// TIA Portal project "ContainerProduction_V0.1.0" (V18)

(* hardware
DEVICE "S7-1500/ET200MP station_1"  S7-1500 station
   slot 0: "Rail_0"  Rack  6ES7 590-1***0-0AA0
   slot 1: "PLC_1"  CPU 1511C-1 PN  6ES7 511-1CK01-0AB0  V2.9
      slot 3: "CPU display_1"  6ES7591-1AA00-0AA0
      slot 32768: "PROFINET interface_1"  X1
         slot 32769: "Port_1"  X1 P1
         slot 32770: "Port_2"  X1 P2
      slot 34817: "Virtual CP interface port_1"  Virtual CP interface port  Virtual CP interface port
*)

// ===== PLC "PLC_1"  CPU 1511C-1 PN =====

VAR_GLOBAL   // PLC tag table "Default tag table"
   "start_btn_sim" AT %M501.0 : Bool;
   "stp_btn_sim" AT %M501.1 : Bool;
   "monitor1 state value" AT %MW2 : UInt;
   "Spare_memory2" AT %M500.2 : Bool;
   "Spare_memory1" AT %M500.3 : Bool;
   "Spare_memory3" AT %M500.4 : Bool;
   "Spare_memory5" AT %M500.5 : Bool;
   "Tag_3" AT %M500.6 : Bool;
   "Tag_4" AT %M500.7 : Bool;
   "Tag_5" AT %M500.1 : Bool;
   "Tag_6" AT %M501.2 : Bool;
   "Tag_7" AT %M111.7 : Bool;
   "Tag_8" AT %M856.7 : Bool;
   "Tag_9" AT %M358.7 : Bool;
   "Tag_10" AT %M123.4 : Bool;
   "Clock_Byte" AT %MB0 : Byte;
   "Clock_10Hz" AT %M0.0 : Bool;
   "Clock_5Hz" AT %M0.1 : Bool;
   "Clock_2.5Hz" AT %M0.2 : Bool;
   "Clock_2Hz" AT %M0.3 : Bool;
   "Clock_1.25Hz" AT %M0.4 : Bool;
   "Clock_1Hz" AT %M0.5 : Bool;
   "Clock_0.625Hz" AT %M0.6 : Bool;
   "Clock_0.5Hz" AT %M0.7 : Bool;
   "Tag_1" AT %M525.5 : Bool;
   "index" AT %MW4 : UInt;   // actual array index value
   "Tag_2" AT %M503.7 : Bool;
   "Tag_11" AT %M853.7 : Bool;
   "Tag_12" AT %M853.0 : Bool;
   "Tag_13" AT %M444.0 : Bool;
END_VAR

VAR_GLOBAL   // PLC tag table "IO_List"
   "Start_Button" AT %I10.0 : Bool;
   "Stop_Button" AT %I10.1 : Bool;
   "Emergency_Stop" AT %I10.2 : Bool;
   "Mold_isClosed" AT %I10.3 : Bool;
   "Mold_isOpen" AT %I10.4 : Bool;
   "Product_Ejected" AT %I10.7 : Bool;
   "NextStation_Buffer_Full" AT %I11.0 : Bool;
   "DI_unused1" AT %I11.1 : Bool;
   "Feeder_Start" AT %Q4.0 : Bool;
   "Injection_Start" AT %Q4.1 : Bool;
   "Mold_Close" AT %Q4.2 : Bool;
   "Mold_Open" AT %Q4.3 : Bool;
   "Ejector_Forward" AT %Q4.4 : Bool;
   "Ejector_Backward" AT %Q4.5 : Bool;
   "Heater_Enable" AT %Q4.6 : Bool;
   "Cooling_Enable" AT %Q4.7 : Bool;
   "Alarm_Buzzer" AT %Q5.0 : Bool;
   "Tower_Light_Red" AT %Q5.1 : Bool;
   "Material_ActLevel" AT %IW0 : Word;
   "Temperature_ActLevel" AT %IW2 : Word;
   "Air_Pressure_ActLevel" AT %IW4 : Word;
   "AQ_unused1" AT %QW0 : Word;
   "Ejector_is_atHome" AT %I10.5 : Bool;
   "Ejector_isExtended" AT %I10.6 : Bool;
   "DI_unused2" AT %I11.2 : Bool;
   "DI_unused3" AT %I11.3 : Bool;
   "DI_unused4" AT %I11.4 : Bool;
   "DI_unused5" AT %I11.5 : Bool;
   "DI_unused6" AT %I11.6 : Bool;
   "DI_unused7" AT %I11.7 : Bool;
   "Tower_Light_Yellow" AT %Q5.2 : Bool;
   "Tower_Light_Green" AT %Q5.3 : Bool;
   "Goto_NextStationBuffer" AT %Q5.4 : Bool;
   "DQ_unused1" AT %Q5.5 : Bool;
   "DQ_unused2" AT %Q5.6 : Bool;
   "DQ_unused3" AT %Q5.7 : Bool;
   "AI_unused1" AT %IW6 : Word;
   "AI_unused2" AT %IW8 : Word;
   "AQ_unused2" AT %QW2 : Word;
END_VAR

// folder: Config

DATA_BLOCK "config_parameters"   // DB2
{ S7_Optimized_Access := 'TRUE' }
VERSION : 0.1
   VAR
      Receipe_Parameters : Array[0..100] of Struct
         Heating_Time : Time;
         Cooling_Time : Time;
         Material_Consumption : Real;
         Temperature_SetVal : Real;
         Pressure_SetVal : Real;
      END_STRUCT;
      Station_Parameters : Struct
         Hopper : Struct
            ErrorLimit : Real := 1250.0;
            HighLimit : Real := 1000.0;
            LowLimit : Real := 350.0;
            EmptyLimit : Real := 50.0;
         END_STRUCT;
         Temperature : Struct
            ErrorLimit : Real := 600.0;
            HighLimit : Real := 550.0;
            LowLimit : Real := 400.0;
         END_STRUCT;
         Pressure : Struct
            ErrorLimit : Real := 15.0;
            HighLimit : Real := 13.0;
            LowLimit : Real := 10.0;
         END_STRUCT;
         Timeout : Struct
            Mold : Struct
               Open : Time;
               Close : Time;
            END_STRUCT;
            Ejector : Struct
               Open : Time;
               Close : Time;
            END_STRUCT;
            ProductDetect : Time;
            Transfer : Time;
         END_STRUCT;
      END_STRUCT;
   END_VAR
BEGIN
   Receipe_Parameters[2].Pressure_SetVal := 12.0;
   Receipe_Parameters[2].Temperature_SetVal := 525.0;
   Receipe_Parameters[2].Material_Consumption := 2000.0;
   Receipe_Parameters[1].Pressure_SetVal := 11.5;   // Pressure_SetVal
   Receipe_Parameters[1].Temperature_SetVal := 500.0;   // Temperature_SetVal
   Receipe_Parameters[1].Material_Consumption := 1000.0;   // Material_Consumption
   Receipe_Parameters[1].Cooling_Time := T#7S;   // Cooling_Time
   Receipe_Parameters[2].Cooling_Time := T#13S;
   Receipe_Parameters[1].Heating_Time := T#5S;   // Heating_Time
   Receipe_Parameters[2].Heating_Time := T#10S;
   Receipe_Parameters[0].Heating_Time := T#3S;
   Receipe_Parameters[0].Cooling_Time := T#3S;
   Receipe_Parameters[0].Material_Consumption := 500.0;
   Receipe_Parameters[0].Temperature_SetVal := 450.0;
   Receipe_Parameters[0].Pressure_SetVal := 11.0;
END_DATA_BLOCK

// folder: Flow-1_Checking_Order_Data

DATA_BLOCK "FB_create_serialNo_DB"   // DB8
{ S7_Optimized_Access := 'TRUE' }
VERSION : 0.1
// stored: InstanceOfName FB_create_serialNo
"FB_create_serialNo"
BEGIN
END_DATA_BLOCK

DATA_BLOCK "FB_CheckOrderData_DB"   // DB23
{ S7_Optimized_Access := 'TRUE' }
VERSION : 0.1
// stored: InstanceOfName FB_CheckOrderData
"FB_CheckOrderData"
BEGIN
END_DATA_BLOCK

// folder: Flow-1_Checking_Order_Data/Checking_MES_data

DATA_BLOCK "FB_checking_orderID_DB_1"   // DB12
{ S7_Optimized_Access := 'TRUE' }
VERSION : 0.1
// stored: InstanceOfName FB_checking_orderID
"FB_checking_orderID"
BEGIN
END_DATA_BLOCK

DATA_BLOCK "FB_checking_productID_DB_1"   // DB13
{ S7_Optimized_Access := 'TRUE' }
VERSION : 0.1
// stored: InstanceOfName FB_checking_productID
"FB_checking_productID"
BEGIN
END_DATA_BLOCK

DATA_BLOCK "FB_checking_receipeID_DB_1"   // DB14
{ S7_Optimized_Access := 'TRUE' }
VERSION : 0.1
// stored: InstanceOfName FB_checking_receipeID
"FB_checking_receipeID"
BEGIN
END_DATA_BLOCK

// folder: Flow-2_Checking_Initial_Conditions

DATA_BLOCK "FB_Control_Initial_Conditions_DB"   // DB25
{ S7_Optimized_Access := 'TRUE' }
VERSION : 0.1
// stored: InstanceOfName FB_Control_Initial_Conditions
"FB_Control_Initial_Conditions"
BEGIN
END_DATA_BLOCK

// folder: Flow3_Run_Molding_State

DATA_BLOCK "FB_Start_Molding_State_DB"   // DB11
{ S7_Optimized_Access := 'TRUE' }
VERSION : 0.1
// stored: InstanceOfName FB_Start_Molding_State
"FB_Start_Molding_State"
BEGIN
END_DATA_BLOCK

// folder: Flow4_Finishing_Molding_State

DATA_BLOCK "FB_Finishing_Molding_DB"   // DB15
{ S7_Optimized_Access := 'TRUE' }
VERSION : 0.1
// stored: InstanceOfName FB_Finishing_Molding
"FB_Finishing_Molding"
BEGIN
END_DATA_BLOCK

// folder: Flow5_Checking_Target_Production

DATA_BLOCK "FB_Checking_Target_Production_DB"   // DB16
{ S7_Optimized_Access := 'TRUE' }
VERSION : 0.1
// stored: InstanceOfName FB_Checking_Target_Production
"FB_Checking_Target_Production"
BEGIN
END_DATA_BLOCK

// folder: Machine_transition

DATA_BLOCK "FB_SubTransition_DB"   // DB9
{ S7_Optimized_Access := 'TRUE' }
VERSION : 0.1
// stored: InstanceOfName FB_SubTransition
"FB_SubTransition"
BEGIN
END_DATA_BLOCK

DATA_BLOCK "FB_control_state_transition_DB"   // DB10
{ S7_Optimized_Access := 'TRUE' }
VERSION : 0.1
// stored: InstanceOfName FB_control_state_transition
"FB_control_state_transition"
BEGIN
END_DATA_BLOCK

// folder: Simulation_data

DATA_BLOCK "FB_simulate_digital_input_DB"   // DB7
{ S7_Optimized_Access := 'TRUE' }
VERSION : 0.1
// stored: InstanceOfName FB_simulate_digital_input
"FB_simulate_digital_input"
BEGIN
END_DATA_BLOCK

DATA_BLOCK "Material_ActLevel_Simulation"   // DB18
{ S7_Optimized_Access := 'TRUE' }
VERSION : 0.1
// stored: InstanceOfName FB_simulate_analog_data
"FB_simulate_analog_data"
BEGIN
END_DATA_BLOCK

DATA_BLOCK "Temperature_Act_Level_Simulation"   // DB19
{ S7_Optimized_Access := 'TRUE' }
VERSION : 0.1
// stored: InstanceOfName FB_simulate_analog_data
"FB_simulate_analog_data"
BEGIN
END_DATA_BLOCK

DATA_BLOCK "Pressure_Act_Level_Simulation"   // DB20
{ S7_Optimized_Access := 'TRUE' }
VERSION : 0.1
// stored: InstanceOfName FB_simulate_analog_data
"FB_simulate_analog_data"
BEGIN
END_DATA_BLOCK

DATA_BLOCK "FB_simulate_digital_input_DB_1"   // DB24
{ S7_Optimized_Access := 'TRUE' }
VERSION : 0.1
// stored: InstanceOfName FB_simulate_digital_input
"FB_simulate_digital_input"
BEGIN
END_DATA_BLOCK

// folder: System blocks/Program resources

DATA_BLOCK "IEC_Counter_0_DB"   // DB17
{ S7_Optimized_Access := 'TRUE' }
AUTHOR : Simatic
FAMILY : IEC
NAME : CNTR
VERSION : 1.0
// stored: InstanceOfName IEC_COUNTER
"IEC_COUNTER"
BEGIN
END_DATA_BLOCK

DATA_BLOCK "IEC_Counter_0_DB_1"   // DB21
{ S7_Optimized_Access := 'TRUE' }
AUTHOR : Simatic
FAMILY : IEC
NAME : UCNTR
VERSION : 1.2
// stored: InstanceOfName IEC_UCOUNTER
"IEC_UCOUNTER"
BEGIN
END_DATA_BLOCK

DATA_BLOCK "IEC_Counter_0_DB_2"   // DB22
{ S7_Optimized_Access := 'TRUE' }
AUTHOR : Simatic
FAMILY : IEC
NAME : CNTR
VERSION : 1.0
// stored: InstanceOfName IEC_COUNTER
"IEC_COUNTER"
BEGIN
END_DATA_BLOCK

// folder: Variable

DATA_BLOCK "VAR_input_simulation"   // DB1
{ S7_Optimized_Access := 'TRUE' }
VERSION : 0.1
   VAR
      DI : Struct
         Start_Button : Bool;
         Stop_Button : Bool;
         Emergency_Stop : Bool;
         Mold_isClosed : Bool;
         Mold_isOpen : Bool := true;
         Ejector_is_atHome : Bool := true;
         Ejector_isExtended : Bool;
         Product_Ejected : Bool;
         NextStation_Buffer_Full : Bool;
         DI_unused1 : Bool := true;
         DI_unused2 : Bool := true;
         DI_unused3 : Bool := true;
         DI_unused4 : Bool := true;
         DI_unused5 : Bool := true;
         DI_unused6 : Bool := true;
         DI_unused7 : Bool := true;
      END_STRUCT;
      AI : Struct
         Material_ActLevel : Real;
         Temperature_ActLevel : Real;
         Air_Pressure_ActLevel : Real;
         AI_unused1 : Real;
         AI_unused2 : Real;
      END_STRUCT;
      Man_material_filling : Bool;
   END_VAR
BEGIN
END_DATA_BLOCK

DATA_BLOCK "VAR_Mes_to_ProductionLine"   // DB3
{ S7_Optimized_Access := 'TRUE' }
VERSION : 0.1
   VAR
      is_Order_Valid : Bool;
      Start_Order : Bool;
      received_MES_data : Struct
         OrderID : String := 'ORD-2026-4321';
         ProductID : String := 'CAP-05L';
         ReciepeID : String := 'RCP-001';
         TargetQuantity : UInt := 500;
      END_STRUCT;
      transmit_MES_data : Struct
         ProductInfo : Struct
            OrderID : String;
            ProductID : UInt;
            ReciepeID : UInt;
            TargetQuantity : UInt;
            ProductSerialNo : String;
         END_STRUCT;
         StationInfo : Struct
            StateNo : UInt;
            StateDescription : String;
            ErrorCode : UInt;
            ErrorDescription : String;
            WarningCode : UInt;
            WarninDescription : String;
            TotalProductionTime : Time;
            ProducedCount : UInt;
            OrderCompleted : Bool;
         END_STRUCT;
         ActualMeasurements : Struct
            ActualTemperature : Real;
            ActualPressure : Real;
            ActualHopperWeight : Real;
         END_STRUCT;
      END_STRUCT;
   END_VAR
BEGIN
END_DATA_BLOCK

DATA_BLOCK "VAR_state_machine"   // DB4
{ S7_Optimized_Access := 'TRUE' }
VERSION : 0.1
   VAR
      start_request : Bool;
      stop_request : Bool;
      st_idle : UInt := 0;
      st_checking_order : UInt := 100;
      st_checking_initial_safety : UInt := 200;
      st_running_molding : UInt := 300;
      st_finishing_molding : UInt := 400;
      st_cycle_completed : UInt := 500;
      st_checking_order_target : UInt := 600;
      st_order_finishing : UInt := 700;
      st_fault : UInt := 9999;
      st_machine_state : UInt := 0;
      previous_state_done : Bool;
      st_simulation_timers : Array[0..5] of IEC_TIMER;
   END_VAR
BEGIN
   st_simulation_timers[0].PT := T#2S_500MS;
   st_simulation_timers[1].PT := T#300MS;
   st_simulation_timers[2].PT := T#1s;
END_DATA_BLOCK

DATA_BLOCK "VAR_outputs"   // DB5
{ S7_Optimized_Access := 'TRUE' }
VERSION : 0.1
   VAR
      Feeder_Start : Bool;
      Injection_Start : Bool;
      Mold_Close : Bool;
      Mold_Open : Bool;
      Ejector_Forward : Bool;
      Ejector_Backward : Bool;
      Heater_Enable : Bool;
      Cooling_Enable : Bool;
      Alarm_Buzzer : Bool;
      Tower_Light_Red : Bool;
      Tower_Light_Yellow : Bool;
      Tower_Light_Green : Bool;
      Goto_NextStationBuffer : Bool;
      DQ_unused1 : Bool;
      DQ_unused2 : Bool;
      DQ_unused3 : Bool;
      AQ_unused1 : Real;
      AQ_unused2 : Real;
   END_VAR
BEGIN
END_DATA_BLOCK

DATA_BLOCK "Err_Wrn_list"   // DB6
{ S7_Optimized_Access := 'TRUE' }
VERSION : 0.1
   VAR
      error_active : Bool;
      warning_active : Bool;
      error_value : UInt;
      warning_value : UInt;
      error_list : Array[0..99] of String;
      warning_list : Array[0..99] of String;
   END_VAR
BEGIN
   error_list[0] := 'No Error';   // Emergeny stop is activated
   error_list[1] := 'Stop request is received';   // Mold is open
   error_list[2] := 'Received OrderID is invalid.';   // Material tank is empty
   error_list[3] := 'Received ProductID is invalid.';   // Thermal value is out of range
   error_list[5] := 'Received target production quantity is invalid.';   // Safety gurad is open
   error_list[4] := 'Received ReceipeID is invalid.';   // Pressure value is out of range
   error_list[6] := 'Creating serialNo error';   // Invalid OrderID
   warning_list[0] := 'No Warning';   // Stop request is received
   warning_list[1] := 'Raw material level is low. Feeding in progress.';   // Material level is low
   error_list[7] := 'Raw material level is too high.';   // Invalid ProductID
   error_list[8] := 'Actual Pressure value is low.';   // Invalid ReceipeID
   error_list[9] := 'Actual pressure level is too high.';   // Invalid Quantity
   error_list[10] := 'Mold closing error';
   error_list[11] := 'Ejector is not at home.';
   error_list[12] := 'Next station buffer is full';
   warning_list[2] := 'Raw material level is critic. Feeding in progress.';
   error_list[13] := 'Temperature is too high.';
   error_list[14] := 'Mold opening error';
END_DATA_BLOCK

// folder: (top level)

FUNCTION_BLOCK "backup"   // FB14, LAD
{ S7_Optimized_Access := 'TRUE' }
VERSION : 0.1
   VAR_TEMP
      Act_rcp_data : UInt;
   END_VAR
BEGIN

REGION Network 1 (SCL): Find out actual receipe parameters in config data
   IF "VAR_Mes_to_ProductionLine".transmit_MES_data.ProductInfo.ProductID <> 0 THEN
       IF "VAR_Mes_to_ProductionLine".transmit_MES_data.ProductInfo.ReciepeID <> 0 THEN
           "index" := "VAR_Mes_to_ProductionLine".transmit_MES_data.ProductInfo.ReciepeID - 1;
           //#Act_rcp_data := "config_parameters".Receipe_Parameters["index"];
       END_IF;
   END_IF;
END_REGION

REGION Network 2: Simulate Analog Inputs according to reciepe parameters
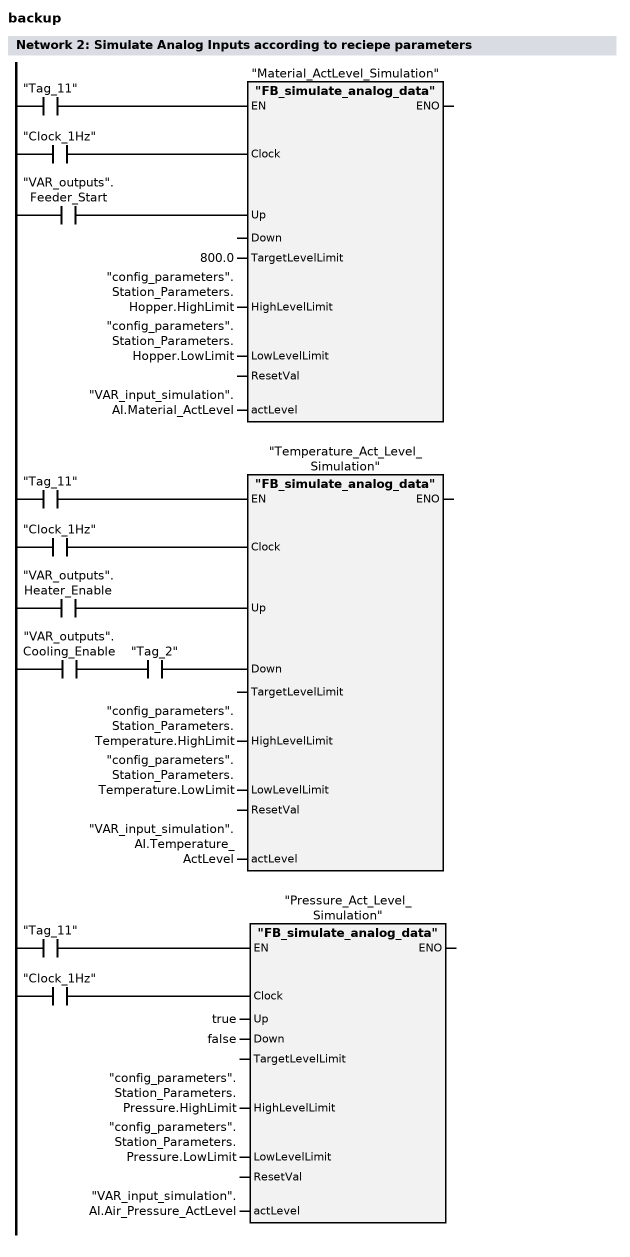
   RUNG wire#powerrail
      Contact( "Tag_11" )
      "Material_ActLevel_Simulation"(Clock := wire#w1, Up := wire#w2, Down :=, TargetLevelLimit := 800.0, HighLevelLimit := "config_parameters".Station_Parameters.Hopper.HighLimit, LowLevelLimit := "config_parameters".Station_Parameters.Hopper.LowLimit, ResetVal :=, actLevel := "VAR_input_simulation".AI.Material_ActLevel)
   END_RUNG
   RUNG wire#powerrail
      Contact( "Clock_1Hz" )
   END_RUNG wire#w1
   RUNG wire#powerrail
      Contact( "VAR_outputs".Feeder_Start )
   END_RUNG wire#w2
   RUNG wire#powerrail
      Contact( "Tag_11" )
      "Temperature_Act_Level_Simulation"(Clock := wire#w3, Up := wire#w4, Down := wire#w5, TargetLevelLimit :=, HighLevelLimit := "config_parameters".Station_Parameters.Temperature.HighLimit, LowLevelLimit := "config_parameters".Station_Parameters.Temperature.LowLimit, ResetVal :=, actLevel := "VAR_input_simulation".AI.Temperature_ActLevel)
   END_RUNG
   RUNG wire#powerrail
      Contact( "Clock_1Hz" )
   END_RUNG wire#w3
   RUNG wire#powerrail
      Contact( "VAR_outputs".Heater_Enable )
   END_RUNG wire#w4
   RUNG wire#powerrail
      Contact( "VAR_outputs".Cooling_Enable )
      Contact( "Tag_2" )
   END_RUNG wire#w5
   RUNG wire#powerrail
      Contact( "Tag_11" )
      "Pressure_Act_Level_Simulation"(Clock := wire#w6, Up := true, Down := false, TargetLevelLimit :=, HighLevelLimit := "config_parameters".Station_Parameters.Pressure.HighLimit, LowLevelLimit := "config_parameters".Station_Parameters.Pressure.LowLimit, ResetVal :=, actLevel := "VAR_input_simulation".AI.Air_Pressure_ActLevel)
   END_RUNG
   RUNG wire#powerrail
      Contact( "Clock_1Hz" )
   END_RUNG wire#w6
   // the same network as SCL:
   IF "Tag_11" THEN
       "Material_ActLevel_Simulation"(Clock := "Clock_1Hz",   // "FB_simulate_analog_data"
                               Up := "VAR_outputs".Feeder_Start,
                               TargetLevelLimit := 800.0,
                               HighLevelLimit := "config_parameters".Station_Parameters.Hopper.HighLimit,
                               LowLevelLimit := "config_parameters".Station_Parameters.Hopper.LowLimit,
                               actLevel := "VAR_input_simulation".AI.Material_ActLevel);
   END_IF;
   IF "Tag_11" THEN
       "Temperature_Act_Level_Simulation"(Clock := "Clock_1Hz",   // "FB_simulate_analog_data"
                               Up := "VAR_outputs".Heater_Enable,
                               Down := "VAR_outputs".Cooling_Enable AND "Tag_2",
                               HighLevelLimit := "config_parameters".Station_Parameters.Temperature.HighLimit,
                               LowLevelLimit := "config_parameters".Station_Parameters.Temperature.LowLimit,
                               actLevel := "VAR_input_simulation".AI.Temperature_ActLevel);
   END_IF;
   IF "Tag_11" THEN
       "Pressure_Act_Level_Simulation"(Clock := "Clock_1Hz",   // "FB_simulate_analog_data"
                               Up := true,
                               Down := false,
                               HighLevelLimit := "config_parameters".Station_Parameters.Pressure.HighLimit,
                               LowLevelLimit := "config_parameters".Station_Parameters.Pressure.LowLimit,
                               actLevel := "VAR_input_simulation".AI.Air_Pressure_ActLevel);
   END_IF;
END_REGION
END_FUNCTION_BLOCK

ORGANIZATION_BLOCK "Main"   // OB1, LAD, ProgramCycle
TITLE = "Main Program Sweep (Cycle)"
{ S7_Optimized_Access := 'TRUE' }
VERSION : 0.1
   VAR_INPUT
      Initial_Call : Bool;   // Initial call of this OB
      Remanence : Bool;   // =True, if remanent data are available
   END_VAR
   VAR_TEMP
      ret_val1 : Int;
      first : DTL;
      ret_val2 : Int;
      second : DTL;
      value : UDInt;
      Act_rcp_data : Struct
         Heating_Time : Time;
         Cooling_Time : Time;
         Material_Consumption : Real;
         Temperature_SetVal : Real;
         Pressure_SetVal : Real;
      END_STRUCT;
   END_VAR
   VAR_TEMP   // added for the SCL form of the ladder/FBD networks
      _w1 : Bool;
   END_VAR
BEGIN

REGION Network 1: Control Start-Stop Request
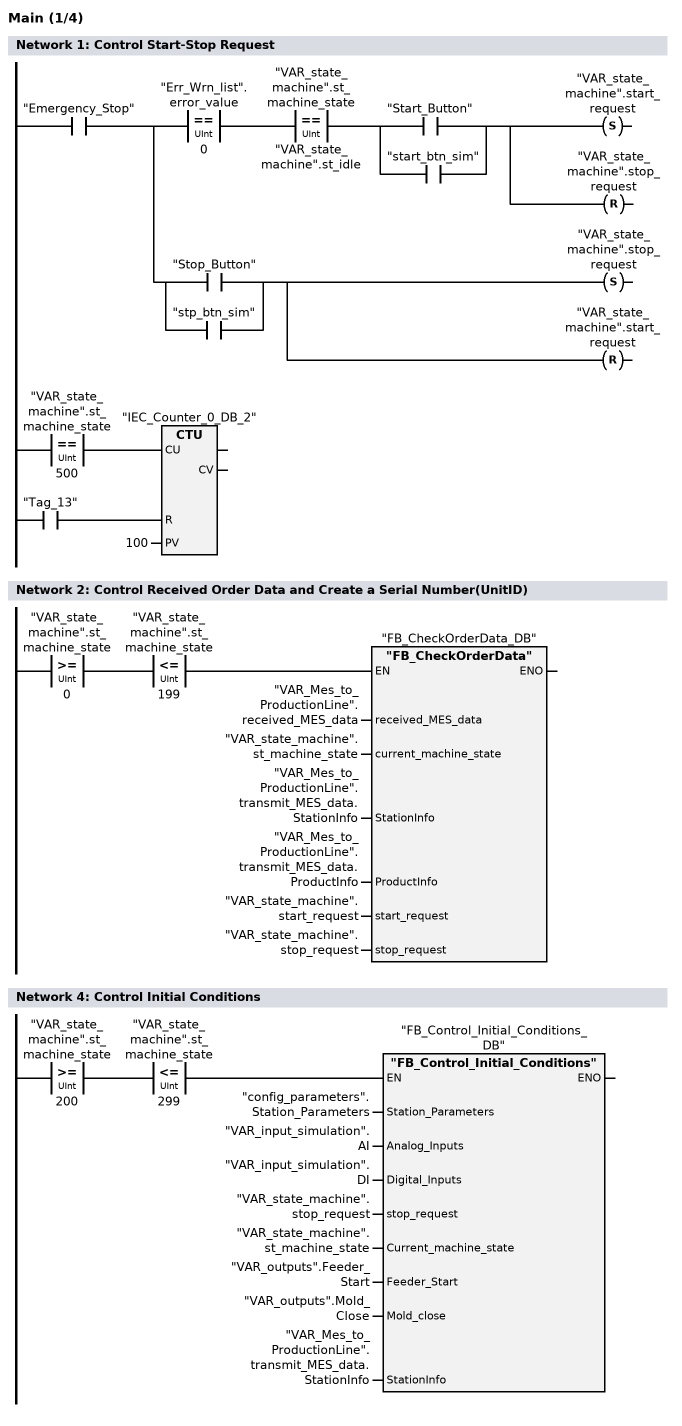
   IF "Emergency_Stop" AND ("Err_Wrn_list".error_value = 0) AND ("VAR_state_machine".st_machine_state = "VAR_state_machine".st_idle) AND ("Start_Button" OR "start_btn_sim") THEN
       "VAR_state_machine".start_request := TRUE;
       "VAR_state_machine".stop_request := FALSE;
   END_IF;
   IF "Emergency_Stop" AND ("Stop_Button" OR "stp_btn_sim") THEN
       "VAR_state_machine".stop_request := TRUE;
       "VAR_state_machine".start_request := FALSE;
   END_IF;
   "IEC_Counter_0_DB_2".CTU(CU := "VAR_state_machine".st_machine_state = 500, R := "Tag_13", PV := 100);
END_REGION

REGION Network 2: Control Received Order Data and Create a Serial Number(UnitID)
   RUNG wire#powerrail
      { S7_Templates := "SrcType := UInt" } GE_Contact(in1 := "VAR_state_machine".st_machine_state, in2 := 0)
      { S7_Templates := "SrcType := UInt" } LE_Contact(in1 := "VAR_state_machine".st_machine_state, in2 := 199)
      "FB_CheckOrderData_DB"(received_MES_data := "VAR_Mes_to_ProductionLine".received_MES_data, current_machine_state := "VAR_state_machine".st_machine_state, StationInfo := "VAR_Mes_to_ProductionLine".transmit_MES_data.StationInfo, ProductInfo := "VAR_Mes_to_ProductionLine".transmit_MES_data.ProductInfo, start_request := "VAR_state_machine".start_request, stop_request := "VAR_state_machine".stop_request)
   END_RUNG
   // the same network as SCL:
   IF ("VAR_state_machine".st_machine_state >= 0) AND ("VAR_state_machine".st_machine_state <= 199) THEN
       "FB_CheckOrderData_DB"(received_MES_data := "VAR_Mes_to_ProductionLine".received_MES_data,   // "FB_CheckOrderData"
                              current_machine_state := "VAR_state_machine".st_machine_state,
                              StationInfo := "VAR_Mes_to_ProductionLine".transmit_MES_data.StationInfo,
                              ProductInfo := "VAR_Mes_to_ProductionLine".transmit_MES_data.ProductInfo,
                              start_request := "VAR_state_machine".start_request,
                              stop_request := "VAR_state_machine".stop_request);
   END_IF;
END_REGION

REGION Network 3 (SCL): Find out actual receipe parameters in config data
   IF "VAR_Mes_to_ProductionLine".transmit_MES_data.ProductInfo.ProductID <> 0 THEN
       IF "VAR_Mes_to_ProductionLine".transmit_MES_data.ProductInfo.ReciepeID <> 0 THEN
           "index" := "VAR_Mes_to_ProductionLine".transmit_MES_data.ProductInfo.ReciepeID - 1;
           #Act_rcp_data := "config_parameters".Receipe_Parameters["index"];
       END_IF;
   END_IF;
END_REGION

REGION Network 4: Control Initial Conditions
   RUNG wire#powerrail
      { S7_Templates := "SrcType := UInt" } GE_Contact(in1 := "VAR_state_machine".st_machine_state, in2 := 200)
      { S7_Templates := "SrcType := UInt" } LE_Contact(in1 := "VAR_state_machine".st_machine_state, in2 := 299)
      "FB_Control_Initial_Conditions_DB"(Station_Parameters := "config_parameters".Station_Parameters, Analog_Inputs := "VAR_input_simulation".AI, Digital_Inputs := "VAR_input_simulation".DI, stop_request := "VAR_state_machine".stop_request, Current_machine_state := "VAR_state_machine".st_machine_state, Feeder_Start := "VAR_outputs".Feeder_Start, Mold_close := "VAR_outputs".Mold_Close, StationInfo := "VAR_Mes_to_ProductionLine".transmit_MES_data.StationInfo)
   END_RUNG
   // the same network as SCL:
   IF ("VAR_state_machine".st_machine_state >= 200) AND ("VAR_state_machine".st_machine_state <= 299) THEN
       "FB_Control_Initial_Conditions_DB"(Station_Parameters := "config_parameters".Station_Parameters,   // "FB_Control_Initial_Conditions"
                               Analog_Inputs := "VAR_input_simulation".AI,
                               Digital_Inputs := "VAR_input_simulation".DI,
                               stop_request := "VAR_state_machine".stop_request,
                               Current_machine_state := "VAR_state_machine".st_machine_state,
                               Feeder_Start := "VAR_outputs".Feeder_Start,
                               Mold_close := "VAR_outputs".Mold_Close,
                               StationInfo := "VAR_Mes_to_ProductionLine".transmit_MES_data.StationInfo);
   END_IF;
END_REGION

REGION Network 5: Run Molding Proccess
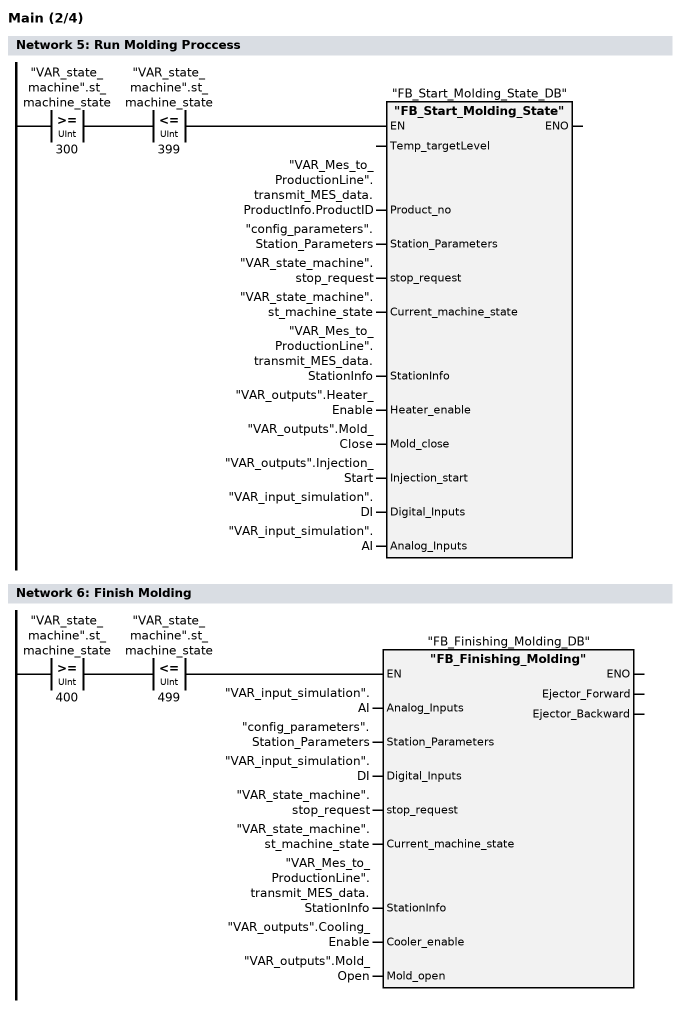
   RUNG wire#powerrail
      { S7_Templates := "SrcType := UInt" } GE_Contact(in1 := "VAR_state_machine".st_machine_state, in2 := 300)
      { S7_Templates := "SrcType := UInt" } LE_Contact(in1 := "VAR_state_machine".st_machine_state, in2 := 399)
      "FB_Start_Molding_State_DB"(Temp_targetLevel :=, Product_no := "VAR_Mes_to_ProductionLine".transmit_MES_data.ProductInfo.ProductID, Station_Parameters := "config_parameters".Station_Parameters, stop_request := "VAR_state_machine".stop_request, Current_machine_state := "VAR_state_machine".st_machine_state, StationInfo := "VAR_Mes_to_ProductionLine".transmit_MES_data.StationInfo, Heater_enable := "VAR_outputs".Heater_Enable, Mold_close := "VAR_outputs".Mold_Close, Injection_start := "VAR_outputs".Injection_Start, Digital_Inputs := "VAR_input_simulation".DI, Analog_Inputs := "VAR_input_simulation".AI)
   END_RUNG
   // the same network as SCL:
   IF ("VAR_state_machine".st_machine_state >= 300) AND ("VAR_state_machine".st_machine_state <= 399) THEN
       "FB_Start_Molding_State_DB"(Product_no := "VAR_Mes_to_ProductionLine".transmit_MES_data.ProductInfo.ProductID,   // "FB_Start_Molding_State"
                               Station_Parameters := "config_parameters".Station_Parameters,
                               stop_request := "VAR_state_machine".stop_request,
                               Current_machine_state := "VAR_state_machine".st_machine_state,
                               StationInfo := "VAR_Mes_to_ProductionLine".transmit_MES_data.StationInfo,
                               Heater_enable := "VAR_outputs".Heater_Enable,
                               Mold_close := "VAR_outputs".Mold_Close,
                               Injection_start := "VAR_outputs".Injection_Start,
                               Digital_Inputs := "VAR_input_simulation".DI,
                               Analog_Inputs := "VAR_input_simulation".AI);
   END_IF;
END_REGION

REGION Network 6: Finish Molding
   RUNG wire#powerrail
      { S7_Templates := "SrcType := UInt" } GE_Contact(in1 := "VAR_state_machine".st_machine_state, in2 := 400)
      { S7_Templates := "SrcType := UInt" } LE_Contact(in1 := "VAR_state_machine".st_machine_state, in2 := 499)
      "FB_Finishing_Molding_DB"(Analog_Inputs := "VAR_input_simulation".AI, Station_Parameters := "config_parameters".Station_Parameters, Digital_Inputs := "VAR_input_simulation".DI, stop_request := "VAR_state_machine".stop_request, Current_machine_state := "VAR_state_machine".st_machine_state, StationInfo := "VAR_Mes_to_ProductionLine".transmit_MES_data.StationInfo, Cooler_enable := "VAR_outputs".Cooling_Enable, Mold_open := "VAR_outputs".Mold_Open, Ejector_Forward =>, Ejector_Backward =>)
   END_RUNG
   // the same network as SCL:
   IF ("VAR_state_machine".st_machine_state >= 400) AND ("VAR_state_machine".st_machine_state <= 499) THEN
       "FB_Finishing_Molding_DB"(Analog_Inputs := "VAR_input_simulation".AI,   // "FB_Finishing_Molding"
                               Station_Parameters := "config_parameters".Station_Parameters,
                               Digital_Inputs := "VAR_input_simulation".DI,
                               stop_request := "VAR_state_machine".stop_request,
                               Current_machine_state := "VAR_state_machine".st_machine_state,
                               StationInfo := "VAR_Mes_to_ProductionLine".transmit_MES_data.StationInfo,
                               Cooler_enable := "VAR_outputs".Cooling_Enable,
                               Mold_open := "VAR_outputs".Mold_Open);
   END_IF;
END_REGION

REGION Network 7: Finish the actual production and check the target quantity
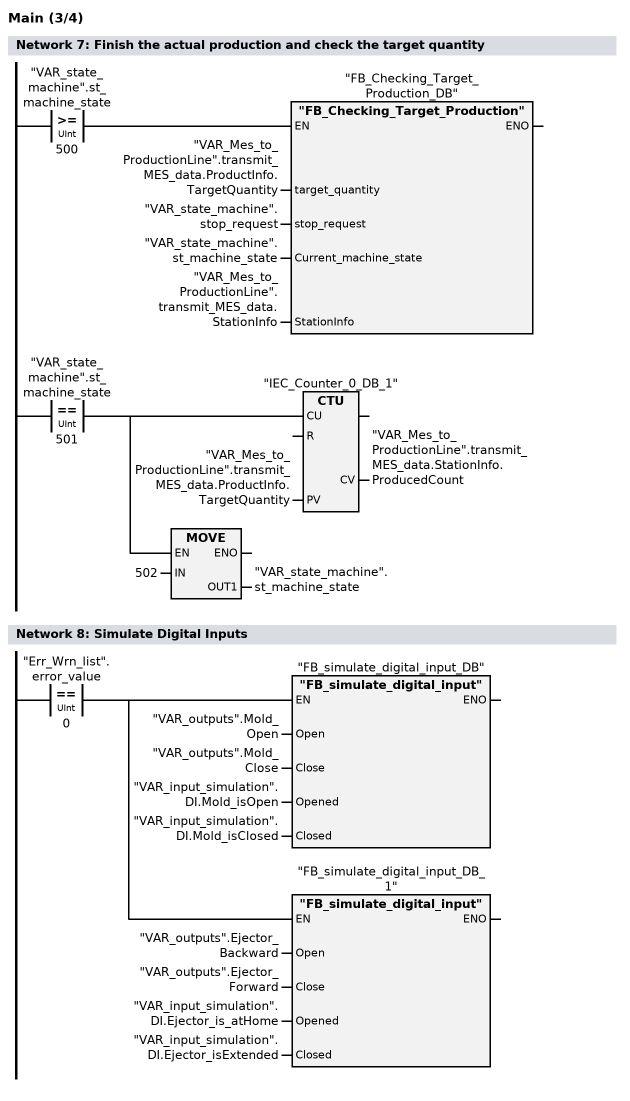
   IF "VAR_state_machine".st_machine_state >= 500 THEN
       "FB_Checking_Target_Production_DB"(target_quantity := "VAR_Mes_to_ProductionLine".transmit_MES_data.ProductInfo.TargetQuantity,   // "FB_Checking_Target_Production"
                               stop_request := "VAR_state_machine".stop_request,
                               Current_machine_state := "VAR_state_machine".st_machine_state,
                               StationInfo := "VAR_Mes_to_ProductionLine".transmit_MES_data.StationInfo);
   END_IF;
   #_w1 := "VAR_state_machine".st_machine_state = 501;
   "IEC_Counter_0_DB_1".CTU(CU := #_w1,
                           PV := "VAR_Mes_to_ProductionLine".transmit_MES_data.ProductInfo.TargetQuantity,
                           CV => "VAR_Mes_to_ProductionLine".transmit_MES_data.StationInfo.ProducedCount);
   IF #_w1 THEN "VAR_state_machine".st_machine_state := 502; END_IF;
END_REGION

REGION Network 8: Simulate Digital Inputs
   RUNG wire#powerrail
      { S7_Templates := "SrcType := UInt" } EQ_Contact(in1 := "Err_Wrn_list".error_value, in2 := 0)
      wire#w1
      "FB_simulate_digital_input_DB"(Open := "VAR_outputs".Mold_Open, Close := "VAR_outputs".Mold_Close, Opened := "VAR_input_simulation".DI.Mold_isOpen, Closed := "VAR_input_simulation".DI.Mold_isClosed)
   END_RUNG
   RUNG wire#w1
      "FB_simulate_digital_input_DB_1"(Open := "VAR_outputs".Ejector_Backward, Close := "VAR_outputs".Ejector_Forward, Opened := "VAR_input_simulation".DI.Ejector_is_atHome, Closed := "VAR_input_simulation".DI.Ejector_isExtended)
   END_RUNG
   // the same network as SCL:
   #_w1 := "Err_Wrn_list".error_value = 0;
   IF #_w1 THEN
       "FB_simulate_digital_input_DB"(Open := "VAR_outputs".Mold_Open,   // "FB_simulate_digital_input"
                               Close := "VAR_outputs".Mold_Close,
                               Opened := "VAR_input_simulation".DI.Mold_isOpen,
                               Closed := "VAR_input_simulation".DI.Mold_isClosed);
       "FB_simulate_digital_input_DB_1"(Open := "VAR_outputs".Ejector_Backward,   // "FB_simulate_digital_input"
                               Close := "VAR_outputs".Ejector_Forward,
                               Opened := "VAR_input_simulation".DI.Ejector_is_atHome,
                               Closed := "VAR_input_simulation".DI.Ejector_isExtended);
   END_IF;
END_REGION

REGION Network 9: Simulate Analog Inputs according to reciepe parameters
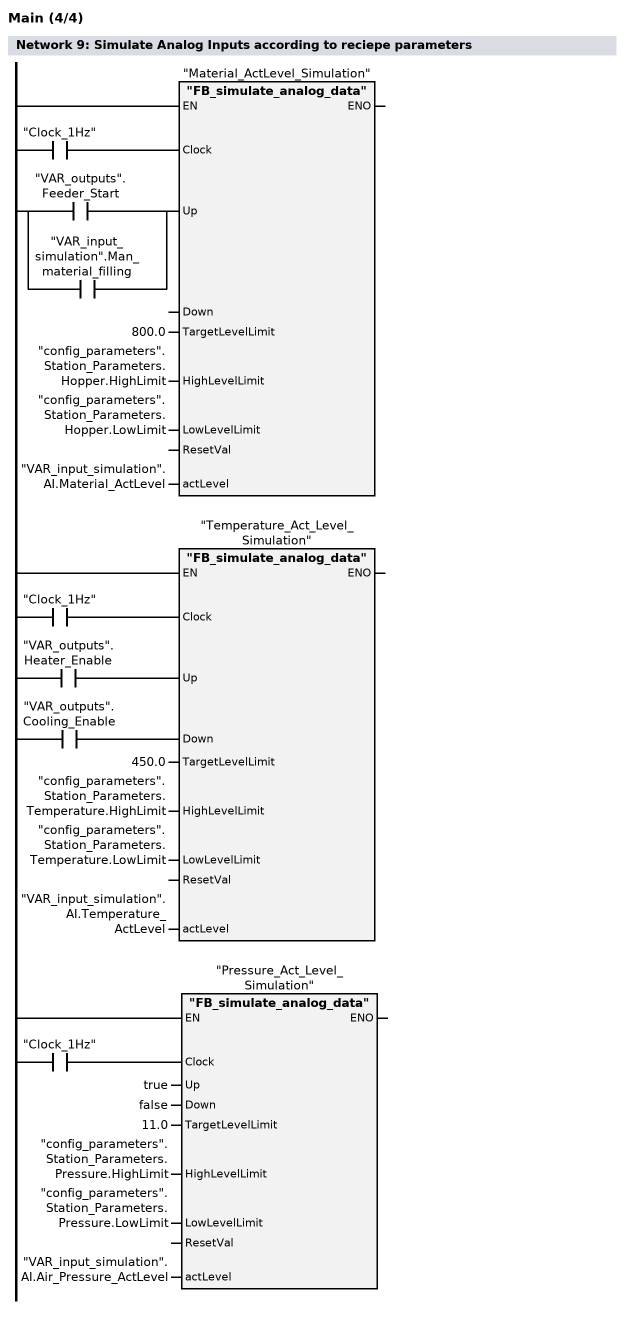
   RUNG wire#powerrail
      "Material_ActLevel_Simulation"(Clock := wire#w1, Up := wire#w2, Down :=, TargetLevelLimit := 800.0, HighLevelLimit := "config_parameters".Station_Parameters.Hopper.HighLimit, LowLevelLimit := "config_parameters".Station_Parameters.Hopper.LowLimit, ResetVal :=, actLevel := "VAR_input_simulation".AI.Material_ActLevel)
   END_RUNG
   RUNG wire#powerrail
      Contact( "Clock_1Hz" )
   END_RUNG wire#w1
   RUNG wire#powerrail
      Contact( "VAR_outputs".Feeder_Start )
   END_RUNG wire#w2
   RUNG wire#powerrail
      Contact( "VAR_input_simulation".Man_material_filling )
   END_RUNG wire#w2
   RUNG wire#powerrail
      "Temperature_Act_Level_Simulation"(Clock := wire#w3, Up := wire#w4, Down := wire#w5, TargetLevelLimit := 450.0, HighLevelLimit := "config_parameters".Station_Parameters.Temperature.HighLimit, LowLevelLimit := "config_parameters".Station_Parameters.Temperature.LowLimit, ResetVal :=, actLevel := "VAR_input_simulation".AI.Temperature_ActLevel)
   END_RUNG
   RUNG wire#powerrail
      Contact( "Clock_1Hz" )
   END_RUNG wire#w3
   RUNG wire#powerrail
      Contact( "VAR_outputs".Heater_Enable )
   END_RUNG wire#w4
   RUNG wire#powerrail
      Contact( "VAR_outputs".Cooling_Enable )
   END_RUNG wire#w5
   RUNG wire#powerrail
      "Pressure_Act_Level_Simulation"(Clock := wire#w6, Up := true, Down := false, TargetLevelLimit := 11.0, HighLevelLimit := "config_parameters".Station_Parameters.Pressure.HighLimit, LowLevelLimit := "config_parameters".Station_Parameters.Pressure.LowLimit, ResetVal :=, actLevel := "VAR_input_simulation".AI.Air_Pressure_ActLevel)
   END_RUNG
   RUNG wire#powerrail
      Contact( "Clock_1Hz" )
   END_RUNG wire#w6
   // the same network as SCL:
   "Material_ActLevel_Simulation"(Clock := "Clock_1Hz",   // "FB_simulate_analog_data"
                           Up := "VAR_outputs".Feeder_Start OR "VAR_input_simulation".Man_material_filling,
                           TargetLevelLimit := 800.0,
                           HighLevelLimit := "config_parameters".Station_Parameters.Hopper.HighLimit,
                           LowLevelLimit := "config_parameters".Station_Parameters.Hopper.LowLimit,
                           actLevel := "VAR_input_simulation".AI.Material_ActLevel);
   "Temperature_Act_Level_Simulation"(Clock := "Clock_1Hz",   // "FB_simulate_analog_data"
                           Up := "VAR_outputs".Heater_Enable,
                           Down := "VAR_outputs".Cooling_Enable,
                           TargetLevelLimit := 450.0,
                           HighLevelLimit := "config_parameters".Station_Parameters.Temperature.HighLimit,
                           LowLevelLimit := "config_parameters".Station_Parameters.Temperature.LowLimit,
                           actLevel := "VAR_input_simulation".AI.Temperature_ActLevel);
   "Pressure_Act_Level_Simulation"(Clock := "Clock_1Hz",   // "FB_simulate_analog_data"
                           Up := true,
                           Down := false,
                           TargetLevelLimit := 11.0,
                           HighLevelLimit := "config_parameters".Station_Parameters.Pressure.HighLimit,
                           LowLevelLimit := "config_parameters".Station_Parameters.Pressure.LowLimit,
                           actLevel := "VAR_input_simulation".AI.Air_Pressure_ActLevel);
END_REGION
END_ORGANIZATION_BLOCK

// folder: Flow-1_Checking_Order_Data

FUNCTION_BLOCK "FB_create_serialNo"   // FB9, SCL
{ S7_Optimized_Access := 'TRUE' }
VERSION : 0.1
   VAR_INPUT
      ProductID : String;
      Year : UInt;
      Month : UInt;
      Day : UInt;
      TimeStamp : UDInt;
   END_VAR
   VAR_OUTPUT
      SerialNo : String;
      Creation_OK : Bool;
   END_VAR
   VAR_TEMP
      Count : USInt;
      String_data : Struct
         Year_strg : String;
         Month_strg : String;
         Day_strg : String;
         Timestamp_strg : String;
      END_STRUCT;
   END_VAR
BEGIN
   //Convert time data to string values

   //year
    VAL_STRG(IN:=#Year,
            SIZE:=4,//year data consist of 4 digits
            PREC:=0,//return integer value
            FORMAT:=16#0001,//put the value at the left
            P:=1,//start digit value
            OUT=>#String_data.Year_strg);

   //month
   VAL_STRG(IN:=#Month,
       SIZE:=2,//month data consist of 2 digits
       PREC:=0,//return integer value
       FORMAT:=16#0001,//put the value at the left
       P:=1,//start digit value
       OUT=>#String_data.Month_strg);

   //day
   VAL_STRG(IN := #Day,
            SIZE := 2,//day data consist of 2 digits
            PREC := 0,//return integer value
            FORMAT := 16#0001,//put the value at the left
            P := 1,//start digit value
            OUT => #String_data.Day_strg);

   //nanosecond
   VAL_STRG(IN := #TimeStamp,
           SIZE := 10,// consist of 10 digits
            PREC := 0,//return integer value
            FORMAT := 16#0001,//put the value at the left
            P := 1,//start digit value
            OUT => #String_data.Timestamp_strg);

   //Create new serial number
   #Count := 0;
   #SerialNo := CONCAT(IN1 := #ProductID, IN2 := '-');
   #SerialNo := CONCAT(IN1 := #SerialNo, IN2 := #String_data.Year_strg);
   #SerialNo := CONCAT(IN1 := #SerialNo, IN2 := #String_data.Month_strg);
   #SerialNo := CONCAT(IN1 := #SerialNo, IN2 := #String_data.Day_strg);
   #SerialNo := CONCAT(IN1 := #SerialNo, IN2 := '-');
   #SerialNo := CONCAT(IN1 := #SerialNo, IN2 := #String_data.Timestamp_strg);

   IF LEN(#SerialNo) > 17 THEN
       #Creation_OK := true;
   ELSE
       #Creation_OK := false;
   END_IF;
END_FUNCTION_BLOCK

FUNCTION_BLOCK "FB_CheckOrderData"   // FB15, LAD
{ S7_Optimized_Access := 'TRUE' }
VERSION : 0.1
   VAR_INPUT
      received_MES_data : Struct
         OrderID : String;
         ProductID : String;
         ReceipeID : String;
         Quantity : UInt;
      END_STRUCT;
   END_VAR
   VAR_IN_OUT
      current_machine_state : UInt;
      StationInfo : Struct
         StateNo : UInt;
         StateDescription : String;
         ErrorCode : UInt;
         ErrorDescription : String;
         WarningCode : UInt;
         WarninDescription : String;
         TotalProductionTime : Time;
         ProducedCount : UInt;
         OrderCompleted : Bool;
      END_STRUCT;
      ProductInfo : Struct
         OrderID : String;
         ProductID : UInt;
         ReciepeID : UInt;
         TargetQuantity : UInt;
         ProductSerialNo : String;
      END_STRUCT;
      start_request : Bool;
      stop_request : Bool;
   END_VAR
   VAR
      process_simulators : Array[0..20] of IEC_TIMER;
      temp_state : UInt;
      error_code : Bool;
      warning_code : Bool;
      year : UInt;
      month : UInt;
      day : UInt;
      timeStamp : UDInt;
      gettingTimeError : Int;
      aux_var1 : Bool;
      aux_var2 : Bool;
      count : Int;
   END_VAR
   VAR CONSTANT
      st_idle : UInt := 0;
      st_checking_order : UInt := 100;
      st_checking_order_sub1 : UInt := 101;
      st_checking_order_sub2 : UInt := 102;
      st_checking_order_sub3 : UInt := 103;
      st_checking_order_sub4 : UInt := 104;
      st_checking_order_sub5 : UInt := 105;
      st_checking_initial_safety : UInt := 200;
   END_VAR
   VAR_TEMP   // added for the SCL form of the ladder/FBD networks
      _w1 : Bool;
      _w2 : Bool;
      _w3 : Bool;
      _w4 : Bool;
      _w5 : Bool;
   END_VAR
BEGIN

REGION Network 1: Control Start Request
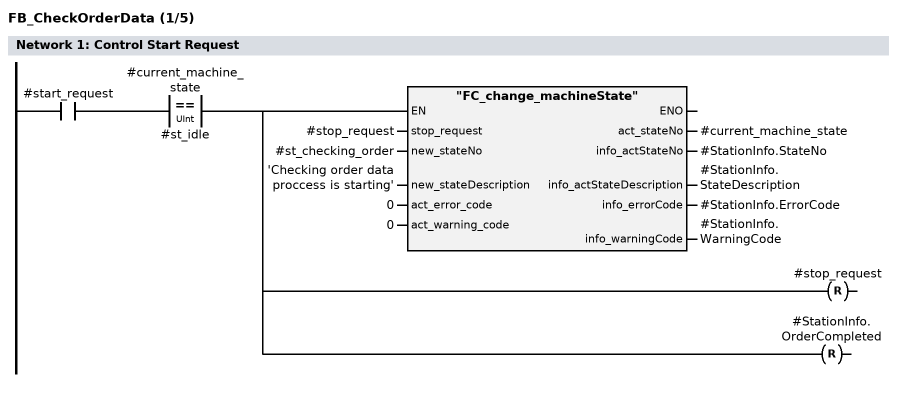
   RUNG wire#powerrail
      Contact( #start_request )
      { S7_Templates := "SrcType := UInt" } EQ_Contact(in1 := #current_machine_state, in2 := #st_idle)
      wire#w1
      "FC_change_machineState"(stop_request := #stop_request, new_stateNo := #st_checking_order, new_stateDescription := 'Checking order data proccess is starting', act_error_code := 0, act_warning_code := 0, act_stateNo => #current_machine_state, info_actStateNo => #StationInfo.StateNo, info_actStateDescription => #StationInfo.StateDescription, info_errorCode => #StationInfo.ErrorCode, info_warningCode => #StationInfo.WarningCode)
   END_RUNG
   RUNG wire#w1
      R_Coil( #stop_request )
   END_RUNG
   RUNG wire#w1
      R_Coil( #StationInfo.OrderCompleted )
   END_RUNG
   // the same network as SCL:
   #_w1 := #start_request AND (#current_machine_state = #st_idle);
   IF #_w1 THEN
       "FC_change_machineState"(stop_request := #stop_request,
                               new_stateNo := #st_checking_order,
                               new_stateDescription := 'Checking order data proccess is starting',
                               act_error_code := 0,
                               act_warning_code := 0,
                               act_stateNo => #current_machine_state,
                               info_actStateNo => #StationInfo.StateNo,
                               info_actStateDescription => #StationInfo.StateDescription,
                               info_errorCode => #StationInfo.ErrorCode,
                               info_warningCode => #StationInfo.WarningCode);
       #stop_request := FALSE;
       #StationInfo.OrderCompleted := FALSE;
   END_IF;
END_REGION

REGION Network 2: Reading and Parsing Received Order Data
   // OrderID : ORD-xxxx-xxxx - String
   // ProductID : CAP-xxL - String
   // ReceipeID : RCP-xxx - String
   // Quantity : Any - Uint
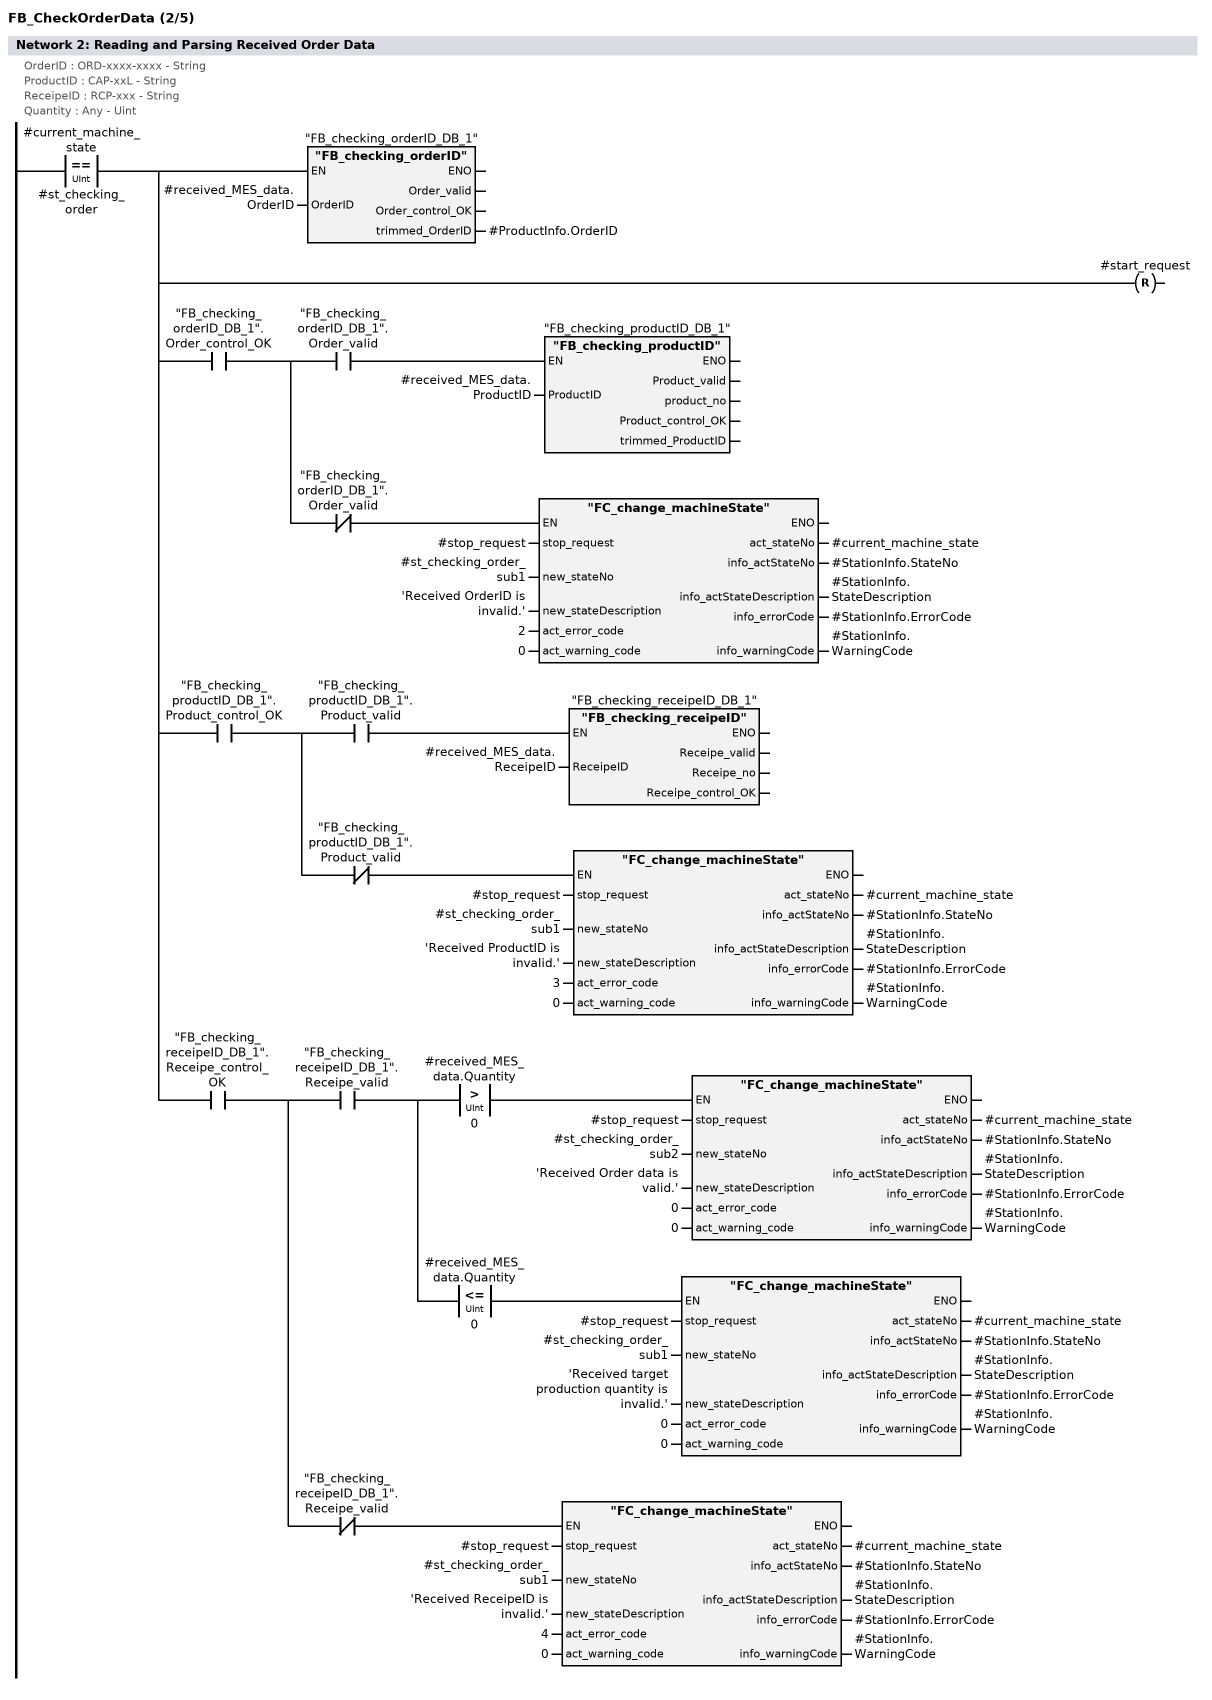
   RUNG wire#powerrail
      { S7_Templates := "SrcType := UInt" } EQ_Contact(in1 := #current_machine_state, in2 := #st_checking_order)
      wire#w1
      "FB_checking_orderID_DB_1"(OrderID := #received_MES_data.OrderID, Order_valid =>, Order_control_OK =>, trimmed_OrderID => #ProductInfo.OrderID)
   END_RUNG
   RUNG wire#w1
      R_Coil( #start_request )
   END_RUNG
   RUNG wire#w1
      Contact( "FB_checking_orderID_DB_1".Order_control_OK )
      wire#w2
      Contact( "FB_checking_orderID_DB_1".Order_valid )
      "FB_checking_productID_DB_1"(ProductID := #received_MES_data.ProductID, Product_valid =>, product_no =>, Product_control_OK =>, trimmed_ProductID =>)
   END_RUNG
   RUNG wire#w2
      I_Contact( "FB_checking_orderID_DB_1".Order_valid )
      "FC_change_machineState"(stop_request := #stop_request, new_stateNo := #st_checking_order_sub1, new_stateDescription := 'Received OrderID is invalid.', act_error_code := 2, act_warning_code := 0, act_stateNo => #current_machine_state, info_actStateNo => #StationInfo.StateNo, info_actStateDescription => #StationInfo.StateDescription, info_errorCode => #StationInfo.ErrorCode, info_warningCode => #StationInfo.WarningCode)
   END_RUNG
   RUNG wire#w1
      Contact( "FB_checking_productID_DB_1".Product_control_OK )
      wire#w3
      Contact( "FB_checking_productID_DB_1".Product_valid )
      "FB_checking_receipeID_DB_1"(ReceipeID := #received_MES_data.ReceipeID, Receipe_valid =>, Receipe_no =>, Receipe_control_OK =>)
   END_RUNG
   RUNG wire#w3
      I_Contact( "FB_checking_productID_DB_1".Product_valid )
      "FC_change_machineState"(stop_request := #stop_request, new_stateNo := #st_checking_order_sub1, new_stateDescription := 'Received ProductID is invalid.', act_error_code := 3, act_warning_code := 0, act_stateNo => #current_machine_state, info_actStateNo => #StationInfo.StateNo, info_actStateDescription => #StationInfo.StateDescription, info_errorCode => #StationInfo.ErrorCode, info_warningCode => #StationInfo.WarningCode)
   END_RUNG
   RUNG wire#w1
      Contact( "FB_checking_receipeID_DB_1".Receipe_control_OK )
      wire#w4
      Contact( "FB_checking_receipeID_DB_1".Receipe_valid )
      wire#w5
      { S7_Templates := "SrcType := UInt" } GT_Contact(in1 := #received_MES_data.Quantity, in2 := 0)
      "FC_change_machineState"(stop_request := #stop_request, new_stateNo := #st_checking_order_sub2, new_stateDescription := 'Received Order data is valid.', act_error_code := 0, act_warning_code := 0, act_stateNo => #current_machine_state, info_actStateNo => #StationInfo.StateNo, info_actStateDescription => #StationInfo.StateDescription, info_errorCode => #StationInfo.ErrorCode, info_warningCode => #StationInfo.WarningCode)
   END_RUNG
   RUNG wire#w5
      { S7_Templates := "SrcType := UInt" } LE_Contact(in1 := #received_MES_data.Quantity, in2 := 0)
      "FC_change_machineState"(stop_request := #stop_request, new_stateNo := #st_checking_order_sub1, new_stateDescription := 'Received target production quantity is invalid.', act_error_code := 0, act_warning_code := 0, act_stateNo => #current_machine_state, info_actStateNo => #StationInfo.StateNo, info_actStateDescription => #StationInfo.StateDescription, info_errorCode => #StationInfo.ErrorCode, info_warningCode => #StationInfo.WarningCode)
   END_RUNG
   RUNG wire#w4
      I_Contact( "FB_checking_receipeID_DB_1".Receipe_valid )
      "FC_change_machineState"(stop_request := #stop_request, new_stateNo := #st_checking_order_sub1, new_stateDescription := 'Received ReceipeID is invalid.', act_error_code := 4, act_warning_code := 0, act_stateNo => #current_machine_state, info_actStateNo => #StationInfo.StateNo, info_actStateDescription => #StationInfo.StateDescription, info_errorCode => #StationInfo.ErrorCode, info_warningCode => #StationInfo.WarningCode)
   END_RUNG
   // the same network as SCL:
   #_w1 := #current_machine_state = #st_checking_order;
   IF #_w1 THEN
       "FB_checking_orderID_DB_1"(OrderID := #received_MES_data.OrderID, trimmed_OrderID => #ProductInfo.OrderID);   // "FB_checking_orderID"
       #start_request := FALSE;
   END_IF;
   #_w2 := #_w1 AND "FB_checking_orderID_DB_1".Order_control_OK;
   IF #_w2 AND "FB_checking_orderID_DB_1".Order_valid THEN
       "FB_checking_productID_DB_1"(ProductID := #received_MES_data.ProductID);   // "FB_checking_productID"
   END_IF;
   IF #_w2 AND NOT "FB_checking_orderID_DB_1".Order_valid THEN
       "FC_change_machineState"(stop_request := #stop_request,
                               new_stateNo := #st_checking_order_sub1,
                               new_stateDescription := 'Received OrderID is invalid.',
                               act_error_code := 2,
                               act_warning_code := 0,
                               act_stateNo => #current_machine_state,
                               info_actStateNo => #StationInfo.StateNo,
                               info_actStateDescription => #StationInfo.StateDescription,
                               info_errorCode => #StationInfo.ErrorCode,
                               info_warningCode => #StationInfo.WarningCode);
   END_IF;
   #_w3 := #_w1 AND "FB_checking_productID_DB_1".Product_control_OK;
   IF #_w3 AND "FB_checking_productID_DB_1".Product_valid THEN
       "FB_checking_receipeID_DB_1"(ReceipeID := #received_MES_data.ReceipeID);   // "FB_checking_receipeID"
   END_IF;
   IF #_w3 AND NOT "FB_checking_productID_DB_1".Product_valid THEN
       "FC_change_machineState"(stop_request := #stop_request,
                               new_stateNo := #st_checking_order_sub1,
                               new_stateDescription := 'Received ProductID is invalid.',
                               act_error_code := 3,
                               act_warning_code := 0,
                               act_stateNo => #current_machine_state,
                               info_actStateNo => #StationInfo.StateNo,
                               info_actStateDescription => #StationInfo.StateDescription,
                               info_errorCode => #StationInfo.ErrorCode,
                               info_warningCode => #StationInfo.WarningCode);
   END_IF;
   #_w4 := #_w1 AND "FB_checking_receipeID_DB_1".Receipe_control_OK;
   #_w5 := #_w4 AND "FB_checking_receipeID_DB_1".Receipe_valid;
   IF #_w5 AND (#received_MES_data.Quantity > 0) THEN
       "FC_change_machineState"(stop_request := #stop_request,
                               new_stateNo := #st_checking_order_sub2,
                               new_stateDescription := 'Received Order data is valid.',
                               act_error_code := 0,
                               act_warning_code := 0,
                               act_stateNo => #current_machine_state,
                               info_actStateNo => #StationInfo.StateNo,
                               info_actStateDescription => #StationInfo.StateDescription,
                               info_errorCode => #StationInfo.ErrorCode,
                               info_warningCode => #StationInfo.WarningCode);
   END_IF;
   IF #_w5 AND (#received_MES_data.Quantity <= 0) THEN
       "FC_change_machineState"(stop_request := #stop_request,
                               new_stateNo := #st_checking_order_sub1,
                               new_stateDescription := 'Received target production quantity is invalid.',
                               act_error_code := 0,
                               act_warning_code := 0,
                               act_stateNo => #current_machine_state,
                               info_actStateNo => #StationInfo.StateNo,
                               info_actStateDescription => #StationInfo.StateDescription,
                               info_errorCode => #StationInfo.ErrorCode,
                               info_warningCode => #StationInfo.WarningCode);
   END_IF;
   IF #_w4 AND NOT "FB_checking_receipeID_DB_1".Receipe_valid THEN
       "FC_change_machineState"(stop_request := #stop_request,
                               new_stateNo := #st_checking_order_sub1,
                               new_stateDescription := 'Received ReceipeID is invalid.',
                               act_error_code := 4,
                               act_warning_code := 0,
                               act_stateNo => #current_machine_state,
                               info_actStateNo => #StationInfo.StateNo,
                               info_actStateDescription => #StationInfo.StateDescription,
                               info_errorCode => #StationInfo.ErrorCode,
                               info_warningCode => #StationInfo.WarningCode);
   END_IF;
END_REGION

REGION Network 3: An error occured and transition to the clearance data and go back to the idle
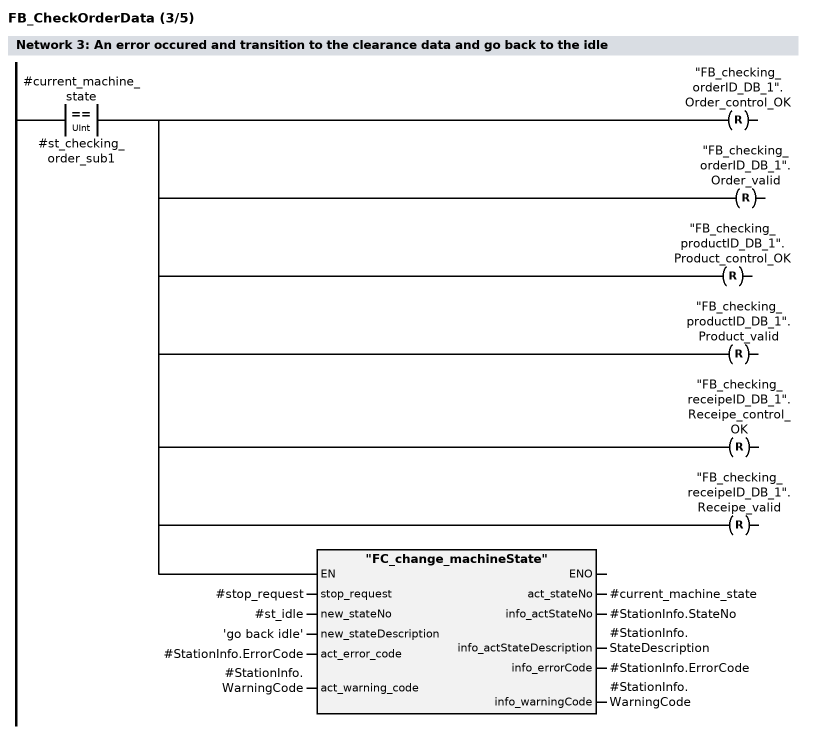
   RUNG wire#powerrail
      { S7_Templates := "SrcType := UInt" } EQ_Contact(in1 := #current_machine_state, in2 := #st_checking_order_sub1)
      wire#w1
      R_Coil( "FB_checking_orderID_DB_1".Order_control_OK )
   END_RUNG
   RUNG wire#w1
      R_Coil( "FB_checking_orderID_DB_1".Order_valid )
   END_RUNG
   RUNG wire#w1
      R_Coil( "FB_checking_productID_DB_1".Product_control_OK )
   END_RUNG
   RUNG wire#w1
      R_Coil( "FB_checking_productID_DB_1".Product_valid )
   END_RUNG
   RUNG wire#w1
      R_Coil( "FB_checking_receipeID_DB_1".Receipe_control_OK )
   END_RUNG
   RUNG wire#w1
      R_Coil( "FB_checking_receipeID_DB_1".Receipe_valid )
   END_RUNG
   RUNG wire#w1
      "FC_change_machineState"(stop_request := #stop_request, new_stateNo := #st_idle, new_stateDescription := 'go back idle', act_error_code := #StationInfo.ErrorCode, act_warning_code := #StationInfo.WarningCode, act_stateNo => #current_machine_state, info_actStateNo => #StationInfo.StateNo, info_actStateDescription => #StationInfo.StateDescription, info_errorCode => #StationInfo.ErrorCode, info_warningCode => #StationInfo.WarningCode)
   END_RUNG
   // the same network as SCL:
   IF #current_machine_state = #st_checking_order_sub1 THEN
       "FB_checking_orderID_DB_1".Order_control_OK := FALSE;
       "FB_checking_orderID_DB_1".Order_valid := FALSE;
       "FB_checking_productID_DB_1".Product_control_OK := FALSE;
       "FB_checking_productID_DB_1".Product_valid := FALSE;
       "FB_checking_receipeID_DB_1".Receipe_control_OK := FALSE;
       "FB_checking_receipeID_DB_1".Receipe_valid := FALSE;
       "FC_change_machineState"(stop_request := #stop_request,
                               new_stateNo := #st_idle,
                               new_stateDescription := 'go back idle',
                               act_error_code := #StationInfo.ErrorCode,
                               act_warning_code := #StationInfo.WarningCode,
                               act_stateNo => #current_machine_state,
                               info_actStateNo => #StationInfo.StateNo,
                               info_actStateDescription => #StationInfo.StateDescription,
                               info_errorCode => #StationInfo.ErrorCode,
                               info_warningCode => #StationInfo.WarningCode);
   END_IF;
END_REGION

REGION Network 4: Create Serial No
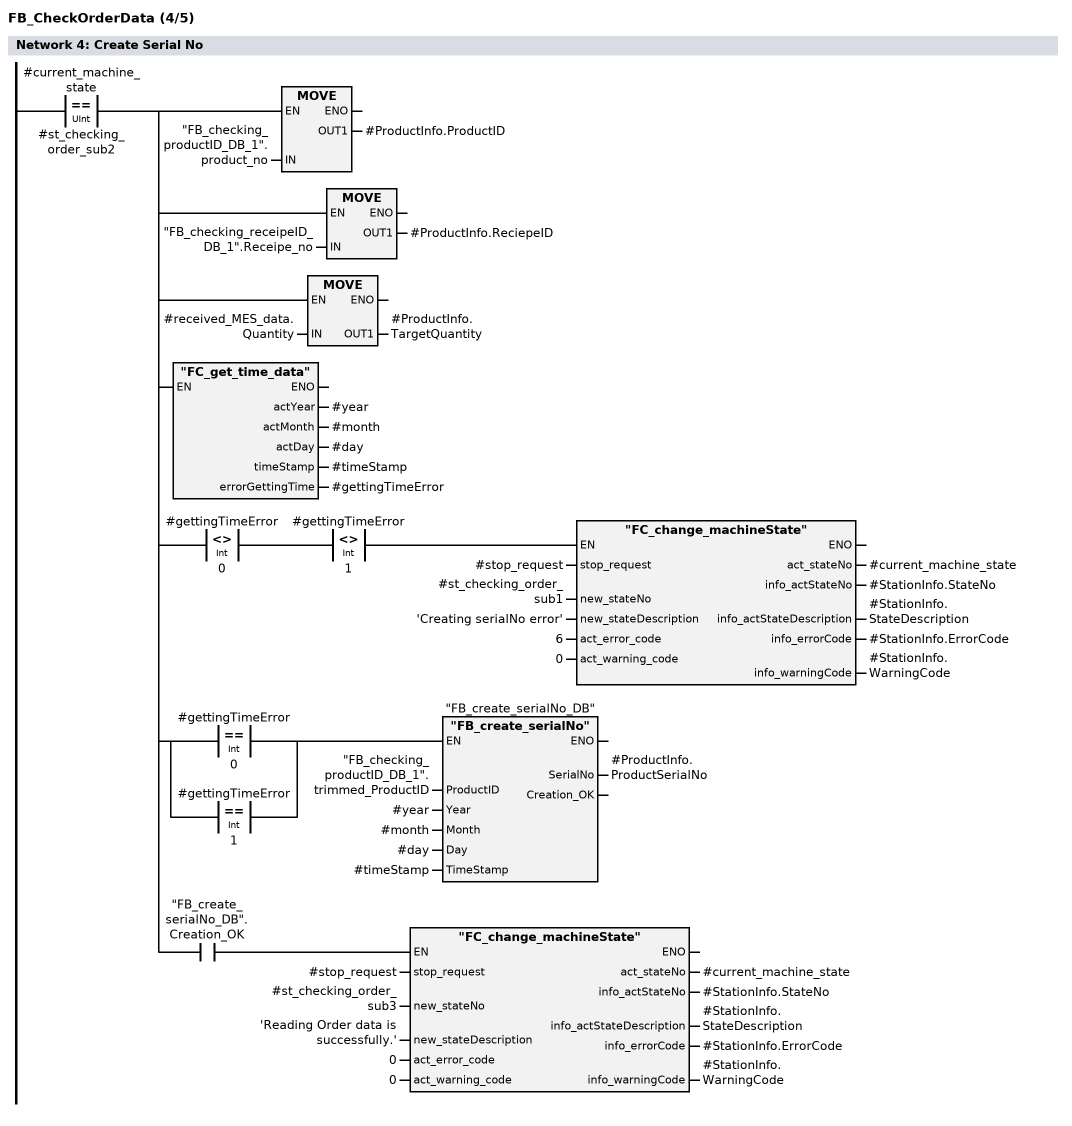
   RUNG wire#powerrail
      { S7_Templates := "SrcType := UInt" } EQ_Contact(in1 := #current_machine_state, in2 := #st_checking_order_sub2)
      wire#w1
      Move(in := "FB_checking_productID_DB_1".product_no, out1 => #ProductInfo.ProductID)
   END_RUNG
   RUNG wire#w1
      Move(in := "FB_checking_receipeID_DB_1".Receipe_no, out1 => #ProductInfo.ReciepeID)
   END_RUNG
   RUNG wire#w1
      Move(in := #received_MES_data.Quantity, out1 => #ProductInfo.TargetQuantity)
   END_RUNG
   RUNG wire#w1
      "FC_get_time_data"(actYear => #year, actMonth => #month, actDay => #day, timeStamp => #timeStamp, errorGettingTime => #gettingTimeError)
   END_RUNG
   RUNG wire#w1
      { S7_Templates := "SrcType := Int" } NE_Contact(in1 := #gettingTimeError, in2 := 0)
      { S7_Templates := "SrcType := Int" } NE_Contact(in1 := #gettingTimeError, in2 := 1)
      "FC_change_machineState"(stop_request := #stop_request, new_stateNo := #st_checking_order_sub1, new_stateDescription := 'Creating serialNo error', act_error_code := 6, act_warning_code := 0, act_stateNo => #current_machine_state, info_actStateNo => #StationInfo.StateNo, info_actStateDescription => #StationInfo.StateDescription, info_errorCode => #StationInfo.ErrorCode, info_warningCode => #StationInfo.WarningCode)
   END_RUNG
   RUNG wire#w1
      { S7_Templates := "SrcType := Int" } EQ_Contact(in1 := #gettingTimeError, in2 := 0)
      wire#w2
      "FB_create_serialNo_DB"(ProductID := "FB_checking_productID_DB_1".trimmed_ProductID, Year := #year, Month := #month, Day := #day, TimeStamp := #timeStamp, SerialNo => #ProductInfo.ProductSerialNo, Creation_OK =>)
   END_RUNG
   RUNG wire#w1
      { S7_Templates := "SrcType := Int" } EQ_Contact(in1 := #gettingTimeError, in2 := 1)
   END_RUNG wire#w2
   RUNG wire#w1
      Contact( "FB_create_serialNo_DB".Creation_OK )
      "FC_change_machineState"(stop_request := #stop_request, new_stateNo := #st_checking_order_sub3, new_stateDescription := 'Reading Order data is successfully.', act_error_code := 0, act_warning_code := 0, act_stateNo => #current_machine_state, info_actStateNo => #StationInfo.StateNo, info_actStateDescription => #StationInfo.StateDescription, info_errorCode => #StationInfo.ErrorCode, info_warningCode => #StationInfo.WarningCode)
   END_RUNG
   // the same network as SCL:
   #_w1 := #current_machine_state = #st_checking_order_sub2;
   IF #_w1 THEN
       #ProductInfo.ProductID := "FB_checking_productID_DB_1".product_no;
       #ProductInfo.ReciepeID := "FB_checking_receipeID_DB_1".Receipe_no;
       #ProductInfo.TargetQuantity := #received_MES_data.Quantity;
       "FC_get_time_data"(actYear => #year,
                          actMonth => #month,
                          actDay => #day,
                          timeStamp => #timeStamp,
                          errorGettingTime => #gettingTimeError);
   END_IF;
   IF #_w1 AND (#gettingTimeError <> 0) AND (#gettingTimeError <> 1) THEN
       "FC_change_machineState"(stop_request := #stop_request,
                               new_stateNo := #st_checking_order_sub1,
                               new_stateDescription := 'Creating serialNo error',
                               act_error_code := 6,
                               act_warning_code := 0,
                               act_stateNo => #current_machine_state,
                               info_actStateNo => #StationInfo.StateNo,
                               info_actStateDescription => #StationInfo.StateDescription,
                               info_errorCode => #StationInfo.ErrorCode,
                               info_warningCode => #StationInfo.WarningCode);
   END_IF;
   IF #_w1 AND ((#gettingTimeError = 0) OR (#gettingTimeError = 1)) THEN
       "FB_create_serialNo_DB"(ProductID := "FB_checking_productID_DB_1".trimmed_ProductID,   // "FB_create_serialNo"
                               Year := #year,
                               Month := #month,
                               Day := #day,
                               TimeStamp := #timeStamp,
                               SerialNo => #ProductInfo.ProductSerialNo);
   END_IF;
   IF #_w1 AND "FB_create_serialNo_DB".Creation_OK THEN
       "FC_change_machineState"(stop_request := #stop_request,
                               new_stateNo := #st_checking_order_sub3,
                               new_stateDescription := 'Reading Order data is successfully.',
                               act_error_code := 0,
                               act_warning_code := 0,
                               act_stateNo => #current_machine_state,
                               info_actStateNo => #StationInfo.StateNo,
                               info_actStateDescription => #StationInfo.StateDescription,
                               info_errorCode => #StationInfo.ErrorCode,
                               info_warningCode => #StationInfo.WarningCode);
   END_IF;
END_REGION

REGION Network 5: Checkink order data step is completed successfully and go to next state
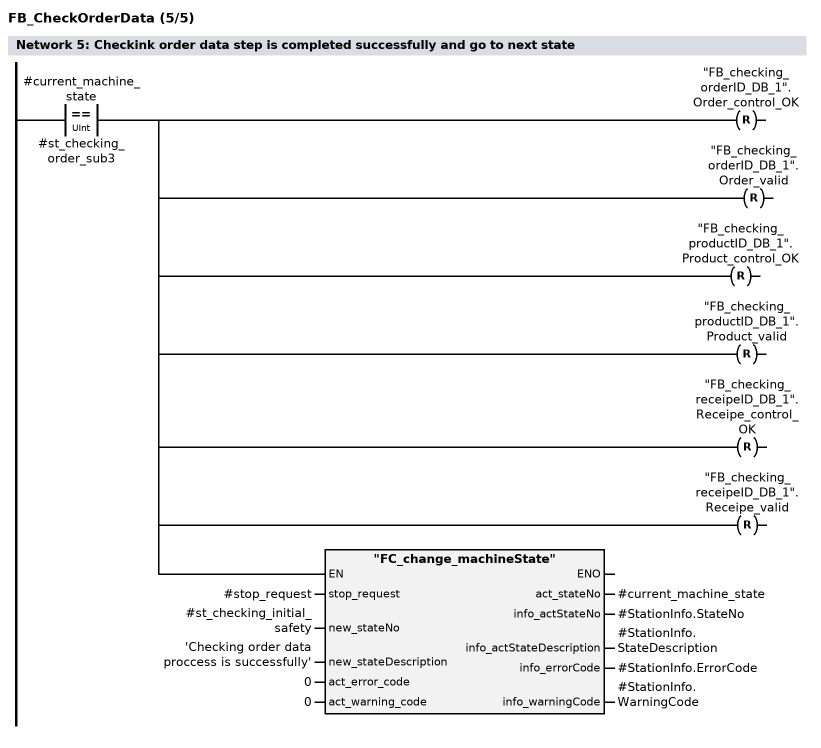
   RUNG wire#powerrail
      { S7_Templates := "SrcType := UInt" } EQ_Contact(in1 := #current_machine_state, in2 := #st_checking_order_sub3)
      wire#w1
      R_Coil( "FB_checking_orderID_DB_1".Order_control_OK )
   END_RUNG
   RUNG wire#w1
      R_Coil( "FB_checking_orderID_DB_1".Order_valid )
   END_RUNG
   RUNG wire#w1
      R_Coil( "FB_checking_productID_DB_1".Product_control_OK )
   END_RUNG
   RUNG wire#w1
      R_Coil( "FB_checking_productID_DB_1".Product_valid )
   END_RUNG
   RUNG wire#w1
      R_Coil( "FB_checking_receipeID_DB_1".Receipe_control_OK )
   END_RUNG
   RUNG wire#w1
      R_Coil( "FB_checking_receipeID_DB_1".Receipe_valid )
   END_RUNG
   RUNG wire#w1
      "FC_change_machineState"(stop_request := #stop_request, new_stateNo := #st_checking_initial_safety, new_stateDescription := 'Checking order data proccess is successfully', act_error_code := 0, act_warning_code := 0, act_stateNo => #current_machine_state, info_actStateNo => #StationInfo.StateNo, info_actStateDescription => #StationInfo.StateDescription, info_errorCode => #StationInfo.ErrorCode, info_warningCode => #StationInfo.WarningCode)
   END_RUNG
   // the same network as SCL:
   IF #current_machine_state = #st_checking_order_sub3 THEN
       "FB_checking_orderID_DB_1".Order_control_OK := FALSE;
       "FB_checking_orderID_DB_1".Order_valid := FALSE;
       "FB_checking_productID_DB_1".Product_control_OK := FALSE;
       "FB_checking_productID_DB_1".Product_valid := FALSE;
       "FB_checking_receipeID_DB_1".Receipe_control_OK := FALSE;
       "FB_checking_receipeID_DB_1".Receipe_valid := FALSE;
       "FC_change_machineState"(stop_request := #stop_request,
                               new_stateNo := #st_checking_initial_safety,
                               new_stateDescription := 'Checking order data proccess is successfully',
                               act_error_code := 0,
                               act_warning_code := 0,
                               act_stateNo => #current_machine_state,
                               info_actStateNo => #StationInfo.StateNo,
                               info_actStateDescription => #StationInfo.StateDescription,
                               info_errorCode => #StationInfo.ErrorCode,
                               info_warningCode => #StationInfo.WarningCode);
   END_IF;
END_REGION
END_FUNCTION_BLOCK

// folder: Flow-1_Checking_Order_Data/Checking_MES_data

FUNCTION_BLOCK "FB_checking_orderID"   // FB1, SCL
{ S7_Optimized_Access := 'TRUE' }
VERSION : 0.1
   VAR_INPUT
      OrderID : String;
   END_VAR
   VAR_OUTPUT
      Order_valid : Bool;
      Order_control_OK : Bool;
      trimmed_OrderID : String;
   END_VAR
   VAR
      simulation_tmr : TON_TIME;
   END_VAR
   VAR_TEMP
      first_index : Int;
      last_index : Int;
      new_orderID : String;
      ID1 : String;
      ID2 : String;
      ID3 : String;
      is_OrderID_Valid : Bool;
      timer_start : Bool;
   END_VAR
   // simulation_tmr.PT := T#5000ms;
BEGIN
   (*
   This function block parses and cleans OrderID received from MES
   *)

   //Check the orderID
   //

   IF LEN(#OrderID) = 0 THEN //invalid OrderID lenght
       #is_OrderID_Valid := FALSE;

   ELSIF LEN(#OrderID) > 0 THEN //valid OrderID lenght
       #first_index := 1;
       #last_index := LEN(#OrderID);

       //Find the index of spaces at the beginning
       WHILE #first_index <= #last_index AND #OrderID[#first_index] = ' ' DO
           #first_index := #first_index + 1;
       END_WHILE;

       //Find the index of spaces at the end
       WHILE #last_index >= #first_index AND #OrderID[#last_index] = ' ' DO
           #last_index := #last_index - 1;
       END_WHILE;

       IF #first_index > #last_index THEN //The orderID consists of only spaces 
           #is_OrderID_Valid := false; //invalid OrderID

       ELSE //trim spaces at the beginnig and end
           #new_orderID := MID(IN := #OrderID, L := (#last_index - #first_index + 1), P := #first_index);
           #trimmed_OrderID := #new_orderID;
       END_IF;

       #ID1 := LEFT(IN := #new_orderID, L := 3); //find and parse 'ORD'
       #ID2 := MID(IN := #new_orderID, L := 4, P := 5); //find and parse the first 'xxxx'. This shows the current year
       #ID3 := RIGHT(IN := #new_orderID, L := 4); //find and parse the second 'xxxx'. This shows the current order number

       IF #ID1 = 'ORD' AND LEN(#ID2) = 4 AND LEN(#ID3) = 4 THEN
           #is_OrderID_Valid := TRUE;
       ELSE
           #is_OrderID_Valid := FALSE;
       END_IF;
   END_IF;



   IF #is_OrderID_Valid THEN
       #Order_valid := true;
       #Order_control_OK := TRUE;
   ELSE
       #Order_valid := false;
       #Order_control_OK := TRUE;
   END_IF;
END_FUNCTION_BLOCK

FUNCTION_BLOCK "FB_checking_receipeID"   // FB2, SCL
{ S7_Optimized_Access := 'TRUE' }
VERSION : 0.1
   VAR_INPUT
      ReceipeID : String;
   END_VAR
   VAR_OUTPUT
      Receipe_valid : Bool;
      Receipe_no : UInt;
      Receipe_control_OK : Bool;
   END_VAR
   VAR_TEMP
      is_ReceipeID_Valid : Bool;
      first_index : Int;
      last_index : Int;
      new_receipeID : String;
      ID1 : String;
      ID2 : String;
      strg_receipe_no : String;
   END_VAR
BEGIN
   (*
   This function block parses and cleans ReceipeID received from MES
   *)

   //Check the ReceipeID
   //

   IF LEN(#ReceipeID) = 0 THEN //invalid ProductID lenght
       #is_ReceipeID_Valid := FALSE;

   ELSIF LEN(#ReceipeID) > 0 THEN //valid ProductID lenght
       #first_index := 1;
       #last_index := LEN(#ReceipeID);

       //Find the index of spaces at the beginning
       WHILE #first_index <= #last_index AND #ReceipeID[#first_index] = ' ' DO
           #first_index := #first_index + 1;
       END_WHILE;

       //Find the index of spaces at the end
       WHILE #last_index >= #first_index AND #ReceipeID[#last_index] = ' ' DO
           #last_index := #last_index - 1;
       END_WHILE;

       IF #first_index > #last_index THEN //The productID consists of only spaces 
           #is_ReceipeID_Valid := false; //invalid OrderID

       ELSE //trim spaces at the beginnig and end
           #new_receipeID := MID(IN := #ReceipeID, L := (#last_index - #first_index + 1), P := #first_index);
       END_IF;

       #ID1 := LEFT(IN := #new_receipeID, L := 3); //find and parse 'RCP'
       #ID2 := RIGHT(IN := #new_receipeID, L := 3); //find and parse the first 'xxx'. This shows the receipe that will be used

       IF #ID1 = 'RCP' AND LEN(#ID2) = 3 THEN

           STRG_VAL(IN := #ID2,
                    FORMAT := 16#0000,
                    P := 1,
                    OUT => #Receipe_no);
           #is_ReceipeID_Valid := TRUE;
       ELSE
           #is_ReceipeID_Valid := FALSE;
       END_IF;
   END_IF;

   IF #is_ReceipeID_Valid THEN
       #Receipe_valid := true;
       #Receipe_control_OK := TRUE;
   ELSE
       #Receipe_valid := false;
       #Receipe_control_OK := TRUE;
   END_IF;
END_FUNCTION_BLOCK

FUNCTION_BLOCK "FB_checking_productID"   // FB5, SCL
{ S7_Optimized_Access := 'TRUE' }
VERSION : 0.1
   VAR_INPUT
      ProductID : String;
   END_VAR
   VAR_OUTPUT
      Product_valid : Bool;
      product_no : UInt;
      Product_control_OK : Bool;
      trimmed_ProductID : String;
   END_VAR
   VAR_TEMP
      is_ProductID_Valid : Bool;
      first_index : Int;
      last_index : Int;
      new_productID : String;
      ID1 : String;
      ID2 : String;
      strg_product_no : String;
   END_VAR
BEGIN
   (*
   This function block parses and cleans ProductID received from MES
   *)

   //Check the ProductID
   //

   IF LEN(#ProductID) = 0 THEN //invalid ProductID lenght
       #is_ProductID_Valid := FALSE;

   ELSIF LEN(#ProductID) > 0 THEN //valid ProductID lenght
       #first_index := 1;
       #last_index := LEN(#ProductID);

       //Find the index of spaces at the beginning
       WHILE #first_index <= #last_index AND #ProductID[#first_index] = ' ' DO
           #first_index := #first_index + 1;
       END_WHILE;

       //Find the index of spaces at the end
       WHILE #last_index >= #first_index AND #ProductID[#last_index] = ' ' DO
           #last_index := #last_index - 1;
       END_WHILE;

       IF #first_index > #last_index THEN //The productID consists of only spaces 
           #is_ProductID_Valid := false; //invalid OrderID

       ELSE //trim spaces at the beginnig and end
           #new_productID := MID(IN := #ProductID, L := (#last_index - #first_index + 1), P := #first_index);
           #trimmed_ProductID := #new_productID;
       END_IF;

       #ID1 := LEFT(IN := #new_productID, L := 3); //find and parse 'CAP'
       #ID2 := RIGHT(IN := #new_productID, L := 3); //find and parse the first 'xxL'. This shows the product no that will be produced

       IF #ID1 = 'CAP' AND LEN(#ID2) = 3 THEN

           #strg_product_no := LEFT(IN := #ID2, L := 2); //find and parse 'CAP'
           STRG_VAL(IN:=#strg_product_no,
                                   FORMAT:=16#0000,
                                   P:=1,
                                   OUT=>#product_no);
           #is_ProductID_Valid := TRUE;
       ELSE
           #is_ProductID_Valid := FALSE;
       END_IF;
   END_IF;

   IF #is_ProductID_Valid THEN
       #Product_valid := true;
       #Product_control_OK := TRUE;
   ELSE
       #Product_valid := false;
       #Product_control_OK := TRUE;
   END_IF;
END_FUNCTION_BLOCK

// folder: Flow-2_Checking_Initial_Conditions

FUNCTION_BLOCK "FB_Control_Initial_Conditions"   // FB4, LAD
{ S7_Optimized_Access := 'TRUE' }
VERSION : 0.1
// In this block, the following steps are executed:
// 
// - Check the material level
// - Check the pressure level
// - Check the positions of the mold actuator and ejector actuator
// - Check if the next station's buffer is empty
   VAR_INPUT
      Station_Parameters : Struct
         Hopper : Struct
            ErrorLimit : Real := 1250.0;
            HighLimit : Real := 1000.0;
            LowLimit : Real := 350.0;
            EmptyLimit : Real := 50.0;
         END_STRUCT;
         Temperature : Struct
            ErrorLimit : Real := 600.0;
            HighLimit : Real := 550.0;
            LowLimit : Real := 400.0;
         END_STRUCT;
         Pressure : Struct
            ErrorLimit : Real := 15.0;
            HighLimit : Real := 13.0;
            LowLimit : Real := 10.0;
         END_STRUCT;
         Timeout : Struct
            Mold : Struct
               Open : Time;
               Close : Time;
            END_STRUCT;
            Ejector : Struct
               Open : Time;
               Close : Time;
            END_STRUCT;
            ProductDetect : Time;
            Transfer : Time;
         END_STRUCT;
      END_STRUCT;
      Analog_Inputs : Struct
         Material_ActLevel : Real;
         Temperature_ActLevel : Real;
         Air_Pressure_ActLevel : Real;
         AI_unused1 : Real;
         AI_unused2 : Real;
      END_STRUCT;
      Digital_Inputs : Struct
         Start_Button : Bool;
         Stop_Button : Bool;
         Emergency_Stop : Bool;
         Mold_isClosed : Bool;
         Mold_isOpen : Bool;
         Ejector_is_atHome : Bool;
         Ejector_isExtended : Bool;
         Product_Ejected : Bool;
         NextStation_Buffer_Full : Bool;
         DI_unused1 : Bool;
         DI_unused2 : Bool;
         DI_unused3 : Bool;
         DI_unused4 : Bool;
         DI_unused5 : Bool;
         DI_unused6 : Bool;
         DI_unused7 : Bool;
      END_STRUCT;
   END_VAR
   VAR_IN_OUT
      stop_request : Bool;
      Current_machine_state : UInt;
      Feeder_Start : Bool;
      Mold_close : Bool;
      StationInfo : Struct
         StateNo : UInt;
         StateDescription : String;
         ErrorCode : UInt;
         ErrorDescription : String;
         WarningCode : UInt;
         WarninDescription : String;
         TotalProductionTime : Time;
         ProducedCount : UInt;
         OrderCompleted : Bool;
      END_STRUCT;
   END_VAR
   VAR
      toplam : UDInt;
      temp_state : UInt;
      aux_var1 : Bool;
      Simulation_Timers : Array[0..10] of IEC_TIMER;
   END_VAR
   VAR_TEMP
      count : Int;
   END_VAR
   VAR CONSTANT
      st_idle : UInt := 0;
      st_checking_order : UInt := 100;
      st_checking_initial_safety : UInt := 200;
      st_checking_initial_safety_sub1 : UInt := 201;
      st_checking_initial_safety_sub2 : UInt := 202;
      st_checking_initial_safety_sub3 : UInt := 203;
      st_checking_initial_safety_sub4 : UInt := 204;
      st_running_molding : UInt := 300;
   END_VAR
   VAR_TEMP   // added for the SCL form of the ladder/FBD networks
      _w1 : Bool;
      _w2 : Bool;
   END_VAR
   // Simulation_Timers[0].PT := T#10S;
BEGIN

REGION Network 1: Checking Material Level and Error Conditions
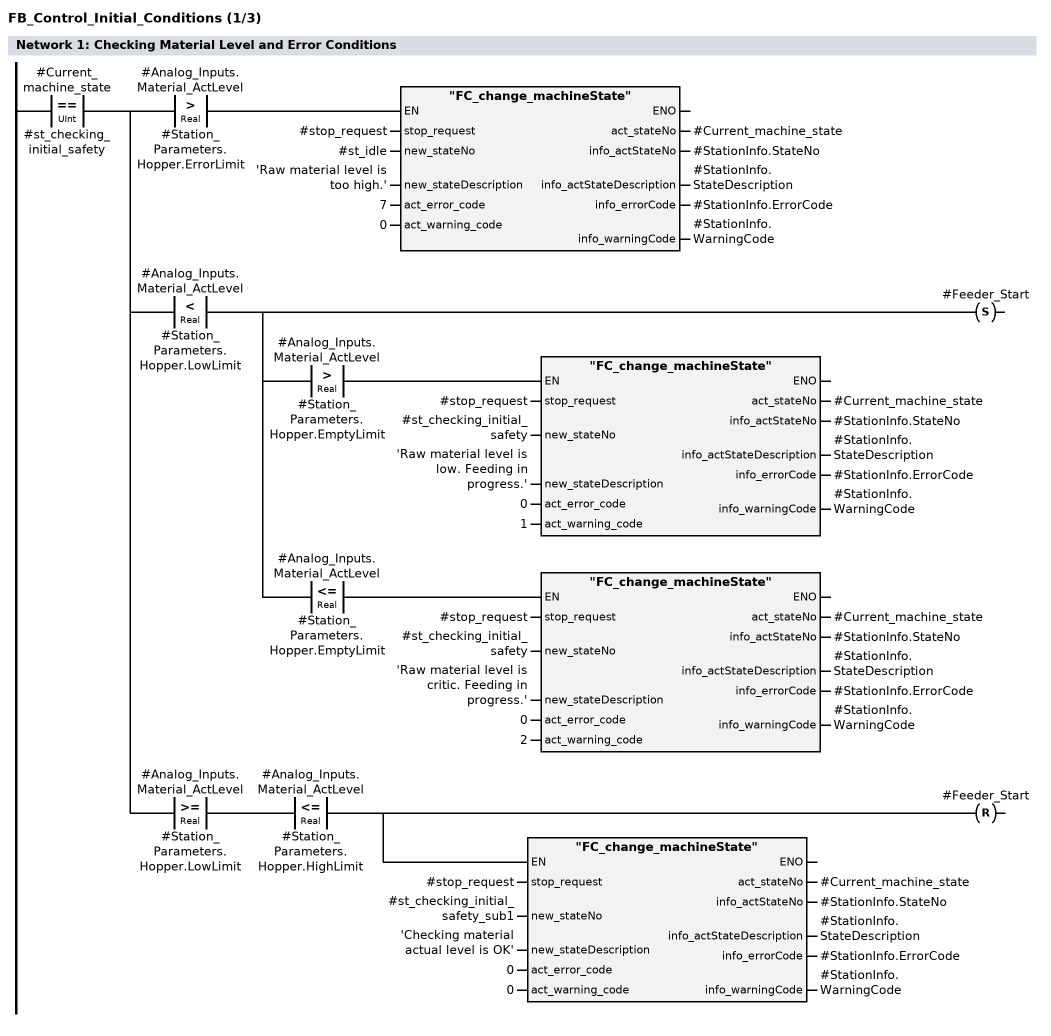
   RUNG wire#powerrail
      { S7_Templates := "SrcType := UInt" } EQ_Contact(in1 := #Current_machine_state, in2 := #st_checking_initial_safety)
      wire#w1
      { S7_Templates := "SrcType := Real" } GT_Contact(in1 := #Analog_Inputs.Material_ActLevel, in2 := #Station_Parameters.Hopper.ErrorLimit)
      "FC_change_machineState"(stop_request := #stop_request, new_stateNo := #st_idle, new_stateDescription := 'Raw material level is too high.', act_error_code := 7, act_warning_code := 0, act_stateNo => #Current_machine_state, info_actStateNo => #StationInfo.StateNo, info_actStateDescription => #StationInfo.StateDescription, info_errorCode => #StationInfo.ErrorCode, info_warningCode => #StationInfo.WarningCode)
   END_RUNG
   RUNG wire#w1
      { S7_Templates := "SrcType := Real" } LT_Contact(in1 := #Analog_Inputs.Material_ActLevel, in2 := #Station_Parameters.Hopper.LowLimit)
      wire#w2
      S_Coil( #Feeder_Start )
   END_RUNG
   RUNG wire#w2
      { S7_Templates := "SrcType := Real" } GT_Contact(in1 := #Analog_Inputs.Material_ActLevel, in2 := #Station_Parameters.Hopper.EmptyLimit)
      "FC_change_machineState"(stop_request := #stop_request, new_stateNo := #st_checking_initial_safety, new_stateDescription := 'Raw material level is low. Feeding in progress.', act_error_code := 0, act_warning_code := 1, act_stateNo => #Current_machine_state, info_actStateNo => #StationInfo.StateNo, info_actStateDescription => #StationInfo.StateDescription, info_errorCode => #StationInfo.ErrorCode, info_warningCode => #StationInfo.WarningCode)
   END_RUNG
   RUNG wire#w2
      { S7_Templates := "SrcType := Real" } LE_Contact(in1 := #Analog_Inputs.Material_ActLevel, in2 := #Station_Parameters.Hopper.EmptyLimit)
      "FC_change_machineState"(stop_request := #stop_request, new_stateNo := #st_checking_initial_safety, new_stateDescription := 'Raw material level is critic. Feeding in progress.', act_error_code := 0, act_warning_code := 2, act_stateNo => #Current_machine_state, info_actStateNo => #StationInfo.StateNo, info_actStateDescription => #StationInfo.StateDescription, info_errorCode => #StationInfo.ErrorCode, info_warningCode => #StationInfo.WarningCode)
   END_RUNG
   RUNG wire#w1
      { S7_Templates := "SrcType := Real" } GE_Contact(in1 := #Analog_Inputs.Material_ActLevel, in2 := #Station_Parameters.Hopper.LowLimit)
      { S7_Templates := "SrcType := Real" } LE_Contact(in1 := #Analog_Inputs.Material_ActLevel, in2 := #Station_Parameters.Hopper.HighLimit)
      wire#w3
      R_Coil( #Feeder_Start )
   END_RUNG
   RUNG wire#w3
      "FC_change_machineState"(stop_request := #stop_request, new_stateNo := #st_checking_initial_safety_sub1, new_stateDescription := 'Checking material actual level is OK', act_error_code := 0, act_warning_code := 0, act_stateNo => #Current_machine_state, info_actStateNo => #StationInfo.StateNo, info_actStateDescription => #StationInfo.StateDescription, info_errorCode => #StationInfo.ErrorCode, info_warningCode => #StationInfo.WarningCode)
   END_RUNG
   // the same network as SCL:
   #_w1 := #Current_machine_state = #st_checking_initial_safety;
   IF #_w1 AND (#Analog_Inputs.Material_ActLevel > #Station_Parameters.Hopper.ErrorLimit) THEN
       "FC_change_machineState"(stop_request := #stop_request,
                               new_stateNo := #st_idle,
                               new_stateDescription := 'Raw material level is too high.',
                               act_error_code := 7,
                               act_warning_code := 0,
                               act_stateNo => #Current_machine_state,
                               info_actStateNo => #StationInfo.StateNo,
                               info_actStateDescription => #StationInfo.StateDescription,
                               info_errorCode => #StationInfo.ErrorCode,
                               info_warningCode => #StationInfo.WarningCode);
   END_IF;
   #_w2 := #_w1 AND (#Analog_Inputs.Material_ActLevel < #Station_Parameters.Hopper.LowLimit);
   IF #_w2 THEN #Feeder_Start := TRUE; END_IF;
   IF #_w2 AND (#Analog_Inputs.Material_ActLevel > #Station_Parameters.Hopper.EmptyLimit) THEN
       "FC_change_machineState"(stop_request := #stop_request,
                               new_stateNo := #st_checking_initial_safety,
                               new_stateDescription := 'Raw material level is low. Feeding in progress.',
                               act_error_code := 0,
                               act_warning_code := 1,
                               act_stateNo => #Current_machine_state,
                               info_actStateNo => #StationInfo.StateNo,
                               info_actStateDescription => #StationInfo.StateDescription,
                               info_errorCode => #StationInfo.ErrorCode,
                               info_warningCode => #StationInfo.WarningCode);
   END_IF;
   IF #_w2 AND (#Analog_Inputs.Material_ActLevel <= #Station_Parameters.Hopper.EmptyLimit) THEN
       "FC_change_machineState"(stop_request := #stop_request,
                               new_stateNo := #st_checking_initial_safety,
                               new_stateDescription := 'Raw material level is critic. Feeding in progress.',
                               act_error_code := 0,
                               act_warning_code := 2,
                               act_stateNo => #Current_machine_state,
                               info_actStateNo => #StationInfo.StateNo,
                               info_actStateDescription => #StationInfo.StateDescription,
                               info_errorCode => #StationInfo.ErrorCode,
                               info_warningCode => #StationInfo.WarningCode);
   END_IF;
   IF #_w1 AND (#Analog_Inputs.Material_ActLevel >= #Station_Parameters.Hopper.LowLimit) AND (#Analog_Inputs.Material_ActLevel <= #Station_Parameters.Hopper.HighLimit) THEN
       #Feeder_Start := FALSE;
       "FC_change_machineState"(stop_request := #stop_request,
                               new_stateNo := #st_checking_initial_safety_sub1,
                               new_stateDescription := 'Checking material actual level is OK',
                               act_error_code := 0,
                               act_warning_code := 0,
                               act_stateNo => #Current_machine_state,
                               info_actStateNo => #StationInfo.StateNo,
                               info_actStateDescription => #StationInfo.StateDescription,
                               info_errorCode => #StationInfo.ErrorCode,
                               info_warningCode => #StationInfo.WarningCode);
   END_IF;
END_REGION

REGION Network 2: Checking Pressure Level and Error Conditions
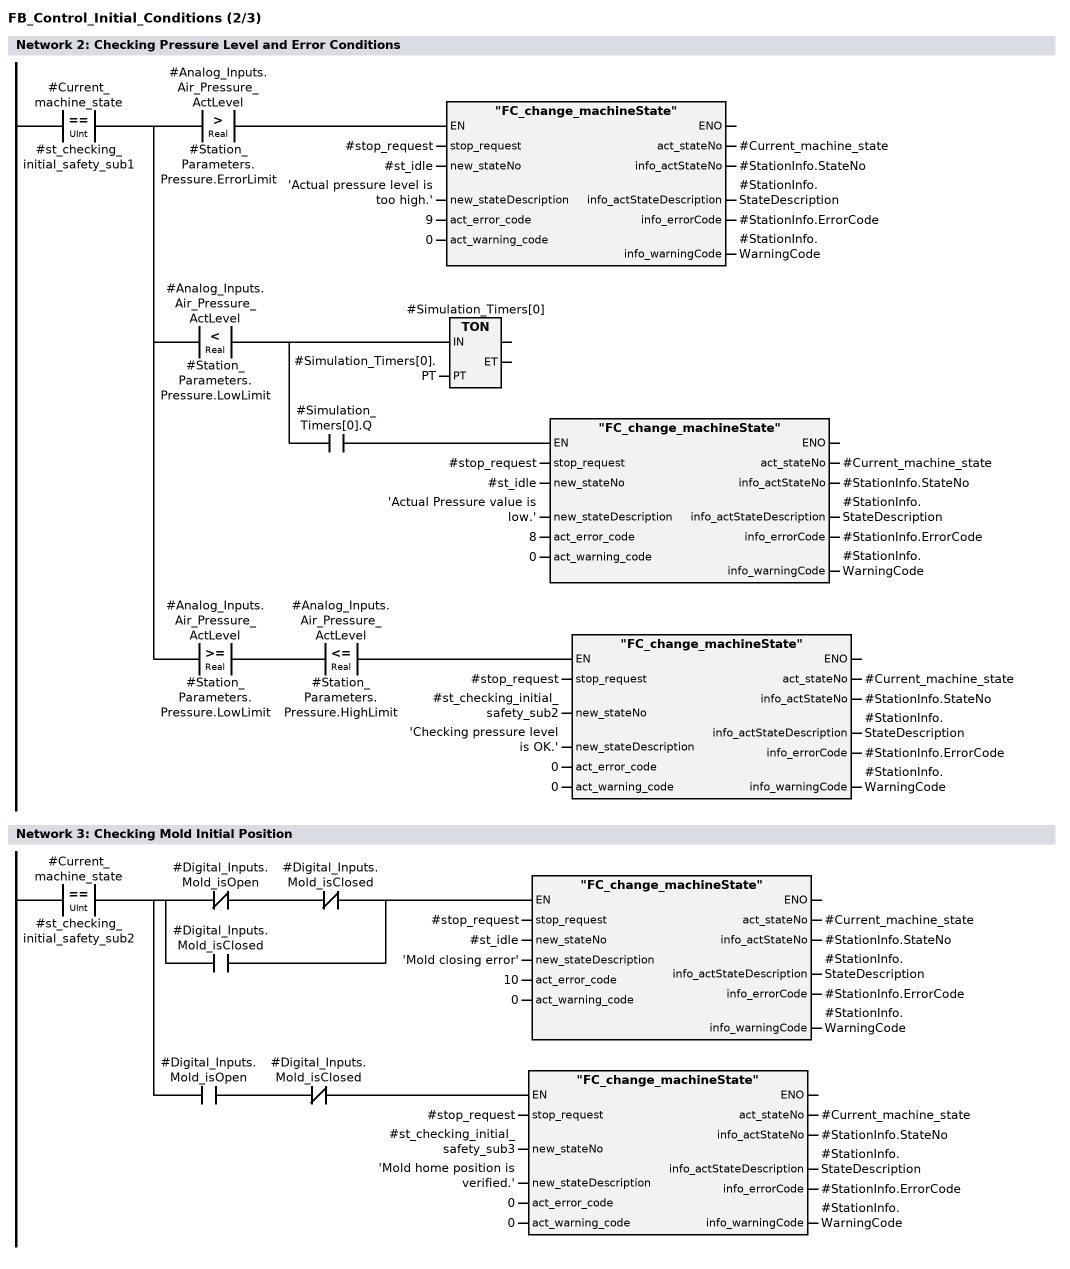
   #_w1 := #Current_machine_state = #st_checking_initial_safety_sub1;
   IF #_w1 AND (#Analog_Inputs.Air_Pressure_ActLevel > #Station_Parameters.Pressure.ErrorLimit) THEN
       "FC_change_machineState"(stop_request := #stop_request,
                               new_stateNo := #st_idle,
                               new_stateDescription := 'Actual pressure level is too high.',
                               act_error_code := 9,
                               act_warning_code := 0,
                               act_stateNo => #Current_machine_state,
                               info_actStateNo => #StationInfo.StateNo,
                               info_actStateDescription => #StationInfo.StateDescription,
                               info_errorCode => #StationInfo.ErrorCode,
                               info_warningCode => #StationInfo.WarningCode);
   END_IF;
   #_w2 := #_w1 AND (#Analog_Inputs.Air_Pressure_ActLevel < #Station_Parameters.Pressure.LowLimit);
   #Simulation_Timers[0].TON(IN := #_w2, PT := #Simulation_Timers[0].PT);
   IF #_w2 AND #Simulation_Timers[0].Q THEN
       "FC_change_machineState"(stop_request := #stop_request,
                               new_stateNo := #st_idle,
                               new_stateDescription := 'Actual Pressure value is low.',
                               act_error_code := 8,
                               act_warning_code := 0,
                               act_stateNo => #Current_machine_state,
                               info_actStateNo => #StationInfo.StateNo,
                               info_actStateDescription => #StationInfo.StateDescription,
                               info_errorCode => #StationInfo.ErrorCode,
                               info_warningCode => #StationInfo.WarningCode);
   END_IF;
   IF #_w1 AND (#Analog_Inputs.Air_Pressure_ActLevel >= #Station_Parameters.Pressure.LowLimit) AND (#Analog_Inputs.Air_Pressure_ActLevel <= #Station_Parameters.Pressure.HighLimit) THEN
       "FC_change_machineState"(stop_request := #stop_request,
                               new_stateNo := #st_checking_initial_safety_sub2,
                               new_stateDescription := 'Checking pressure level is OK.',
                               act_error_code := 0,
                               act_warning_code := 0,
                               act_stateNo => #Current_machine_state,
                               info_actStateNo => #StationInfo.StateNo,
                               info_actStateDescription => #StationInfo.StateDescription,
                               info_errorCode => #StationInfo.ErrorCode,
                               info_warningCode => #StationInfo.WarningCode);
   END_IF;
END_REGION

REGION Network 3: Checking Mold Initial Position
   RUNG wire#powerrail
      { S7_Templates := "SrcType := UInt" } EQ_Contact(in1 := #Current_machine_state, in2 := #st_checking_initial_safety_sub2)
      wire#w1
      I_Contact( #Digital_Inputs.Mold_isOpen )
      I_Contact( #Digital_Inputs.Mold_isClosed )
      wire#w2
      "FC_change_machineState"(stop_request := #stop_request, new_stateNo := #st_idle, new_stateDescription := 'Mold closing error', act_error_code := 10, act_warning_code := 0, act_stateNo => #Current_machine_state, info_actStateNo => #StationInfo.StateNo, info_actStateDescription => #StationInfo.StateDescription, info_errorCode => #StationInfo.ErrorCode, info_warningCode => #StationInfo.WarningCode)
   END_RUNG
   RUNG wire#w1
      Contact( #Digital_Inputs.Mold_isClosed )
   END_RUNG wire#w2
   RUNG wire#w1
      Contact( #Digital_Inputs.Mold_isOpen )
      I_Contact( #Digital_Inputs.Mold_isClosed )
      "FC_change_machineState"(stop_request := #stop_request, new_stateNo := #st_checking_initial_safety_sub3, new_stateDescription := 'Mold home position is verified.', act_error_code := 0, act_warning_code := 0, act_stateNo => #Current_machine_state, info_actStateNo => #StationInfo.StateNo, info_actStateDescription => #StationInfo.StateDescription, info_errorCode => #StationInfo.ErrorCode, info_warningCode => #StationInfo.WarningCode)
   END_RUNG
   // the same network as SCL:
   #_w1 := #Current_machine_state = #st_checking_initial_safety_sub2;
   IF #_w1 AND ((NOT #Digital_Inputs.Mold_isOpen AND NOT #Digital_Inputs.Mold_isClosed) OR #Digital_Inputs.Mold_isClosed) THEN
       "FC_change_machineState"(stop_request := #stop_request,
                               new_stateNo := #st_idle,
                               new_stateDescription := 'Mold closing error',
                               act_error_code := 10,
                               act_warning_code := 0,
                               act_stateNo => #Current_machine_state,
                               info_actStateNo => #StationInfo.StateNo,
                               info_actStateDescription => #StationInfo.StateDescription,
                               info_errorCode => #StationInfo.ErrorCode,
                               info_warningCode => #StationInfo.WarningCode);
   END_IF;
   IF #_w1 AND #Digital_Inputs.Mold_isOpen AND NOT #Digital_Inputs.Mold_isClosed THEN
       "FC_change_machineState"(stop_request := #stop_request,
                               new_stateNo := #st_checking_initial_safety_sub3,
                               new_stateDescription := 'Mold home position is verified.',
                               act_error_code := 0,
                               act_warning_code := 0,
                               act_stateNo => #Current_machine_state,
                               info_actStateNo => #StationInfo.StateNo,
                               info_actStateDescription => #StationInfo.StateDescription,
                               info_errorCode => #StationInfo.ErrorCode,
                               info_warningCode => #StationInfo.WarningCode);
   END_IF;
END_REGION

REGION Network 4: Checking Ejector Initial Position
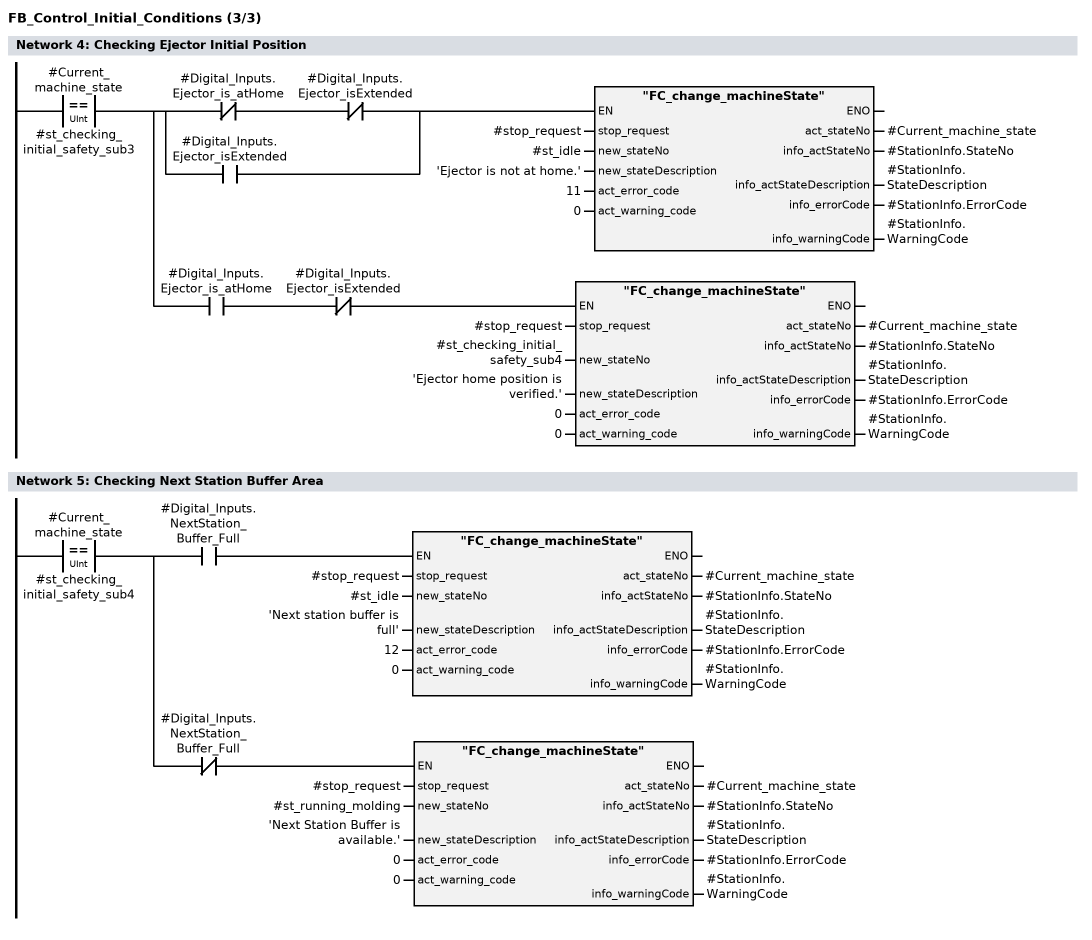
   RUNG wire#powerrail
      { S7_Templates := "SrcType := UInt" } EQ_Contact(in1 := #Current_machine_state, in2 := #st_checking_initial_safety_sub3)
      wire#w1
      I_Contact( #Digital_Inputs.Ejector_is_atHome )
      I_Contact( #Digital_Inputs.Ejector_isExtended )
      wire#w2
      "FC_change_machineState"(stop_request := #stop_request, new_stateNo := #st_idle, new_stateDescription := 'Ejector is not at home.', act_error_code := 11, act_warning_code := 0, act_stateNo => #Current_machine_state, info_actStateNo => #StationInfo.StateNo, info_actStateDescription => #StationInfo.StateDescription, info_errorCode => #StationInfo.ErrorCode, info_warningCode => #StationInfo.WarningCode)
   END_RUNG
   RUNG wire#w1
      Contact( #Digital_Inputs.Ejector_isExtended )
   END_RUNG wire#w2
   RUNG wire#w1
      Contact( #Digital_Inputs.Ejector_is_atHome )
      I_Contact( #Digital_Inputs.Ejector_isExtended )
      "FC_change_machineState"(stop_request := #stop_request, new_stateNo := #st_checking_initial_safety_sub4, new_stateDescription := 'Ejector home position is verified.', act_error_code := 0, act_warning_code := 0, act_stateNo => #Current_machine_state, info_actStateNo => #StationInfo.StateNo, info_actStateDescription => #StationInfo.StateDescription, info_errorCode => #StationInfo.ErrorCode, info_warningCode => #StationInfo.WarningCode)
   END_RUNG
   // the same network as SCL:
   #_w1 := #Current_machine_state = #st_checking_initial_safety_sub3;
   IF #_w1 AND ((NOT #Digital_Inputs.Ejector_is_atHome AND NOT #Digital_Inputs.Ejector_isExtended) OR #Digital_Inputs.Ejector_isExtended) THEN
       "FC_change_machineState"(stop_request := #stop_request,
                               new_stateNo := #st_idle,
                               new_stateDescription := 'Ejector is not at home.',
                               act_error_code := 11,
                               act_warning_code := 0,
                               act_stateNo => #Current_machine_state,
                               info_actStateNo => #StationInfo.StateNo,
                               info_actStateDescription => #StationInfo.StateDescription,
                               info_errorCode => #StationInfo.ErrorCode,
                               info_warningCode => #StationInfo.WarningCode);
   END_IF;
   IF #_w1 AND #Digital_Inputs.Ejector_is_atHome AND NOT #Digital_Inputs.Ejector_isExtended THEN
       "FC_change_machineState"(stop_request := #stop_request,
                               new_stateNo := #st_checking_initial_safety_sub4,
                               new_stateDescription := 'Ejector home position is verified.',
                               act_error_code := 0,
                               act_warning_code := 0,
                               act_stateNo => #Current_machine_state,
                               info_actStateNo => #StationInfo.StateNo,
                               info_actStateDescription => #StationInfo.StateDescription,
                               info_errorCode => #StationInfo.ErrorCode,
                               info_warningCode => #StationInfo.WarningCode);
   END_IF;
END_REGION

REGION Network 5: Checking Next Station Buffer Area
   RUNG wire#powerrail
      { S7_Templates := "SrcType := UInt" } EQ_Contact(in1 := #Current_machine_state, in2 := #st_checking_initial_safety_sub4)
      wire#w1
      Contact( #Digital_Inputs.NextStation_Buffer_Full )
      "FC_change_machineState"(stop_request := #stop_request, new_stateNo := #st_idle, new_stateDescription := 'Next station buffer is full', act_error_code := 12, act_warning_code := 0, act_stateNo => #Current_machine_state, info_actStateNo => #StationInfo.StateNo, info_actStateDescription => #StationInfo.StateDescription, info_errorCode => #StationInfo.ErrorCode, info_warningCode => #StationInfo.WarningCode)
   END_RUNG
   RUNG wire#w1
      I_Contact( #Digital_Inputs.NextStation_Buffer_Full )
      "FC_change_machineState"(stop_request := #stop_request, new_stateNo := #st_running_molding, new_stateDescription := 'Next Station Buffer is available.', act_error_code := 0, act_warning_code := 0, act_stateNo => #Current_machine_state, info_actStateNo => #StationInfo.StateNo, info_actStateDescription => #StationInfo.StateDescription, info_errorCode => #StationInfo.ErrorCode, info_warningCode => #StationInfo.WarningCode)
   END_RUNG
   // the same network as SCL:
   #_w1 := #Current_machine_state = #st_checking_initial_safety_sub4;
   IF #_w1 AND #Digital_Inputs.NextStation_Buffer_Full THEN
       "FC_change_machineState"(stop_request := #stop_request,
                               new_stateNo := #st_idle,
                               new_stateDescription := 'Next station buffer is full',
                               act_error_code := 12,
                               act_warning_code := 0,
                               act_stateNo => #Current_machine_state,
                               info_actStateNo => #StationInfo.StateNo,
                               info_actStateDescription => #StationInfo.StateDescription,
                               info_errorCode => #StationInfo.ErrorCode,
                               info_warningCode => #StationInfo.WarningCode);
   END_IF;
   IF #_w1 AND NOT #Digital_Inputs.NextStation_Buffer_Full THEN
       "FC_change_machineState"(stop_request := #stop_request,
                               new_stateNo := #st_running_molding,
                               new_stateDescription := 'Next Station Buffer is available.',
                               act_error_code := 0,
                               act_warning_code := 0,
                               act_stateNo => #Current_machine_state,
                               info_actStateNo => #StationInfo.StateNo,
                               info_actStateDescription => #StationInfo.StateDescription,
                               info_errorCode => #StationInfo.ErrorCode,
                               info_warningCode => #StationInfo.WarningCode);
   END_IF;
END_REGION
END_FUNCTION_BLOCK

// folder: Flow3_Run_Molding_State

FUNCTION_BLOCK "FB_Start_Molding_State"   // FB7, LAD
{ S7_Optimized_Access := 'TRUE' }
VERSION : 0.1
   VAR_INPUT
      Temp_targetLevel : Real := 450.0;
      Product_no : UInt;
      Station_Parameters : Struct
         Hopper : Struct
            ErrorLimit : Real := 1250.0;
            HighLimit : Real := 1000.0;
            LowLimit : Real := 350.0;
            EmptyLimit : Real := 50.0;
         END_STRUCT;
         Temperature : Struct
            ErrorLimit : Real := 600.0;
            HighLimit : Real := 550.0;
            LowLimit : Real := 400.0;
         END_STRUCT;
         Pressure : Struct
            ErrorLimit : Real := 15.0;
            HighLimit : Real := 13.0;
            LowLimit : Real := 10.0;
         END_STRUCT;
         Timeout : Struct
            Mold : Struct
               Open : Time;
               Close : Time;
            END_STRUCT;
            Ejector : Struct
               Open : Time;
               Close : Time;
            END_STRUCT;
            ProductDetect : Time;
            Transfer : Time;
         END_STRUCT;
      END_STRUCT;
   END_VAR
   VAR_IN_OUT
      stop_request : Bool;
      Current_machine_state : UInt;
      StationInfo : Struct
         StateNo : UInt;
         StateDescription : String;
         ErrorCode : UInt;
         ErrorDescription : String;
         WarningCode : UInt;
         WarninDescription : String;
         TotalProductionTime : Time;
         ProducedCount : UInt;
         OrderCompleted : Bool;
      END_STRUCT;
      Heater_enable : Bool;
      Mold_close : Bool;
      Injection_start : Bool;
      Digital_Inputs : Struct
         Start_Button : Bool;
         Stop_Button : Bool;
         Emergency_Stop : Bool;
         Mold_isClosed : Bool;
         Mold_isOpen : Bool;
         Ejector_is_atHome : Bool;
         Ejector_isExtended : Bool;
         Product_Ejected : Bool;
         NextStation_Buffer_Full : Bool;
         DI_unused1 : Bool;
         DI_unused2 : Bool;
         DI_unused3 : Bool;
         DI_unused4 : Bool;
         DI_unused5 : Bool;
         DI_unused6 : Bool;
         DI_unused7 : Bool;
      END_STRUCT;
      Analog_Inputs : Struct
         Material_ActLevel : Real;
         Temperature_ActLevel : Real;
         Air_Pressure_ActLevel : Real;
         AI_unused1 : Real;
         AI_unused2 : Real;
      END_STRUCT;
   END_VAR
   VAR
      temp_state : UInt;
      Timeout : Array[0..5] of IEC_TIMER;
      Process_Simulation_Timers : Array[0..20] of IEC_TIMER;
      aux_var1 : Bool;
      injection_value : Real;
      injected_value : Real;
   END_VAR
   VAR CONSTANT
      st_idle : UInt := 0;
      st_running_molding : UInt := 300;
      st_running_molding_sub1 : UInt := 301;
      st_running_molding_sub2 : UInt := 302;
      st_running_molding_sub3 : UInt := 303;
      st_running_molding_sub4 : UInt := 304;
      st_running_molding_sub5 : UInt := 305;
      st_running_molding_sub6 : UInt := 306;
      st_finishing_molding : UInt := 400;
      container_05gr : Real := 50.0;
      container_1gr : Real := 100.0;
      container_2gr : Real := 200.0;
   END_VAR
   VAR_TEMP   // added for the SCL form of the ladder/FBD networks
      _w1 : Bool;
      _w2 : Bool;
   END_VAR
   // Process_Simulation_Timers[0].PT := T#500MS;
   // Process_Simulation_Timers[1].PT := T#2S_500MS;
   // Process_Simulation_Timers[2].PT := T#300MS;
   // Process_Simulation_Timers[3].PT := T#10S;
BEGIN

REGION Network 1: Start Heating Process - Check Actual Temperature Value and Control Heater
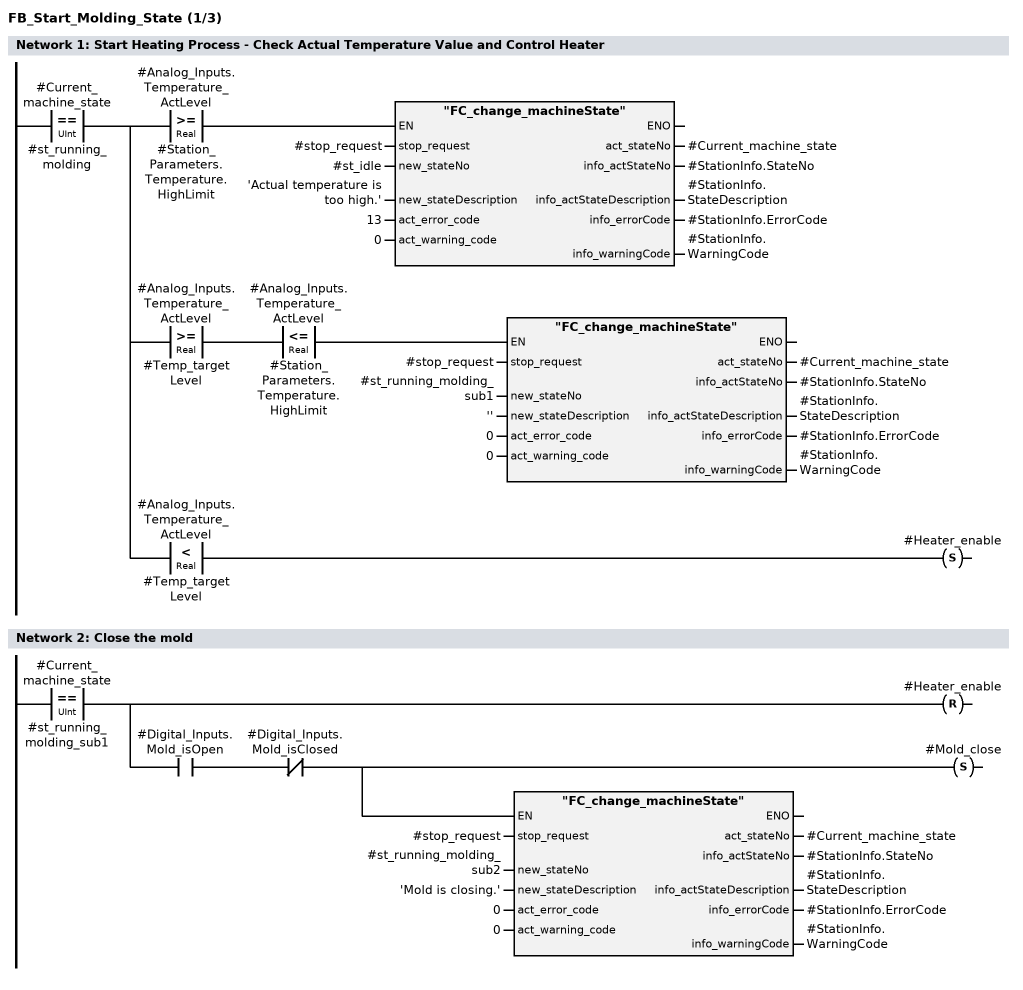
   RUNG wire#powerrail
      { S7_Templates := "SrcType := UInt" } EQ_Contact(in1 := #Current_machine_state, in2 := #st_running_molding)
      wire#w1
      { S7_Templates := "SrcType := Real" } GE_Contact(in1 := #Analog_Inputs.Temperature_ActLevel, in2 := #Station_Parameters.Temperature.HighLimit)
      "FC_change_machineState"(stop_request := #stop_request, new_stateNo := #st_idle, new_stateDescription := 'Actual temperature is too high.', act_error_code := 13, act_warning_code := 0, act_stateNo => #Current_machine_state, info_actStateNo => #StationInfo.StateNo, info_actStateDescription => #StationInfo.StateDescription, info_errorCode => #StationInfo.ErrorCode, info_warningCode => #StationInfo.WarningCode)
   END_RUNG
   RUNG wire#w1
      { S7_Templates := "SrcType := Real" } GE_Contact(in1 := #Analog_Inputs.Temperature_ActLevel, in2 := #Temp_targetLevel)
      { S7_Templates := "SrcType := Real" } LE_Contact(in1 := #Analog_Inputs.Temperature_ActLevel, in2 := #Station_Parameters.Temperature.HighLimit)
      "FC_change_machineState"(stop_request := #stop_request, new_stateNo := #st_running_molding_sub1, new_stateDescription := '', act_error_code := 0, act_warning_code := 0, act_stateNo => #Current_machine_state, info_actStateNo => #StationInfo.StateNo, info_actStateDescription => #StationInfo.StateDescription, info_errorCode => #StationInfo.ErrorCode, info_warningCode => #StationInfo.WarningCode)
   END_RUNG
   RUNG wire#w1
      { S7_Templates := "SrcType := Real" } LT_Contact(in1 := #Analog_Inputs.Temperature_ActLevel, in2 := #Temp_targetLevel)
      S_Coil( #Heater_enable )
   END_RUNG
   // the same network as SCL:
   #_w1 := #Current_machine_state = #st_running_molding;
   IF #_w1 AND (#Analog_Inputs.Temperature_ActLevel >= #Station_Parameters.Temperature.HighLimit) THEN
       "FC_change_machineState"(stop_request := #stop_request,
                               new_stateNo := #st_idle,
                               new_stateDescription := 'Actual temperature is too high.',
                               act_error_code := 13,
                               act_warning_code := 0,
                               act_stateNo => #Current_machine_state,
                               info_actStateNo => #StationInfo.StateNo,
                               info_actStateDescription => #StationInfo.StateDescription,
                               info_errorCode => #StationInfo.ErrorCode,
                               info_warningCode => #StationInfo.WarningCode);
   END_IF;
   IF #_w1 AND (#Analog_Inputs.Temperature_ActLevel >= #Temp_targetLevel) AND (#Analog_Inputs.Temperature_ActLevel <= #Station_Parameters.Temperature.HighLimit) THEN
       "FC_change_machineState"(stop_request := #stop_request,
                               new_stateNo := #st_running_molding_sub1,
                               new_stateDescription := '',
                               act_error_code := 0,
                               act_warning_code := 0,
                               act_stateNo => #Current_machine_state,
                               info_actStateNo => #StationInfo.StateNo,
                               info_actStateDescription => #StationInfo.StateDescription,
                               info_errorCode => #StationInfo.ErrorCode,
                               info_warningCode => #StationInfo.WarningCode);
   END_IF;
   IF #_w1 AND (#Analog_Inputs.Temperature_ActLevel < #Temp_targetLevel) THEN #Heater_enable := TRUE; END_IF;
END_REGION

REGION Network 2: Close the mold
   RUNG wire#powerrail
      { S7_Templates := "SrcType := UInt" } EQ_Contact(in1 := #Current_machine_state, in2 := #st_running_molding_sub1)
      wire#w1
      R_Coil( #Heater_enable )
   END_RUNG
   RUNG wire#w1
      Contact( #Digital_Inputs.Mold_isOpen )
      I_Contact( #Digital_Inputs.Mold_isClosed )
      wire#w2
      S_Coil( #Mold_close )
   END_RUNG
   RUNG wire#w2
      "FC_change_machineState"(stop_request := #stop_request, new_stateNo := #st_running_molding_sub2, new_stateDescription := 'Mold is closing.', act_error_code := 0, act_warning_code := 0, act_stateNo => #Current_machine_state, info_actStateNo => #StationInfo.StateNo, info_actStateDescription => #StationInfo.StateDescription, info_errorCode => #StationInfo.ErrorCode, info_warningCode => #StationInfo.WarningCode)
   END_RUNG
   // the same network as SCL:
   #_w1 := #Current_machine_state = #st_running_molding_sub1;
   IF #_w1 THEN #Heater_enable := FALSE; END_IF;
   IF #_w1 AND #Digital_Inputs.Mold_isOpen AND NOT #Digital_Inputs.Mold_isClosed THEN
       #Mold_close := TRUE;
       "FC_change_machineState"(stop_request := #stop_request,
                               new_stateNo := #st_running_molding_sub2,
                               new_stateDescription := 'Mold is closing.',
                               act_error_code := 0,
                               act_warning_code := 0,
                               act_stateNo => #Current_machine_state,
                               info_actStateNo => #StationInfo.StateNo,
                               info_actStateDescription => #StationInfo.StateDescription,
                               info_errorCode => #StationInfo.ErrorCode,
                               info_warningCode => #StationInfo.WarningCode);
   END_IF;
END_REGION

REGION Network 3
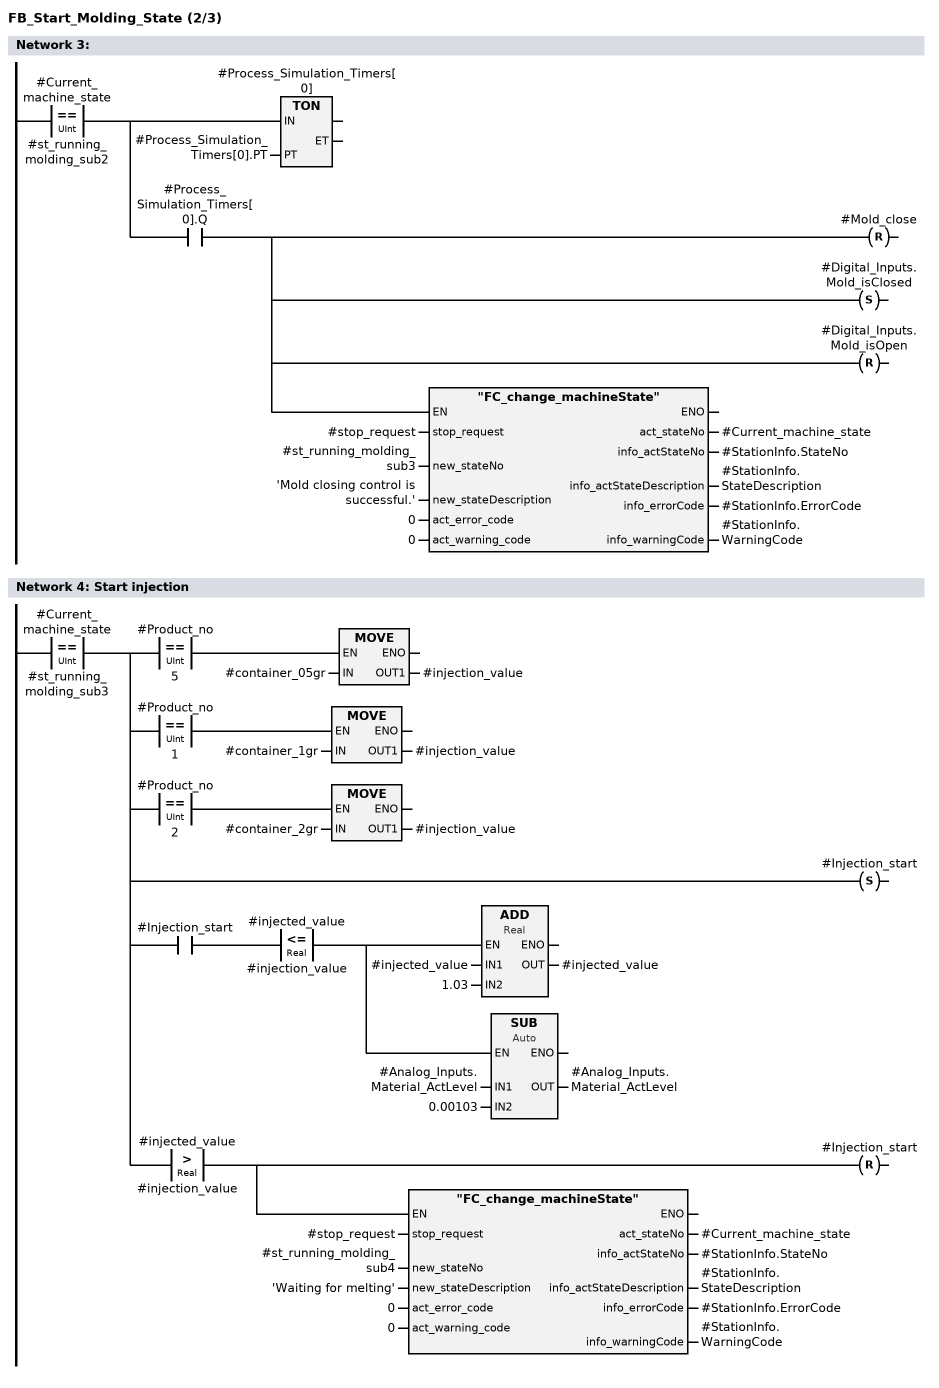
   #_w1 := #Current_machine_state = #st_running_molding_sub2;
   #Process_Simulation_Timers[0].TON(IN := #_w1, PT := #Process_Simulation_Timers[0].PT);
   IF #_w1 AND #Process_Simulation_Timers[0].Q THEN
       #Mold_close := FALSE;
       #Digital_Inputs.Mold_isClosed := TRUE;
       #Digital_Inputs.Mold_isOpen := FALSE;
       "FC_change_machineState"(stop_request := #stop_request,
                               new_stateNo := #st_running_molding_sub3,
                               new_stateDescription := 'Mold closing control is successful.',
                               act_error_code := 0,
                               act_warning_code := 0,
                               act_stateNo => #Current_machine_state,
                               info_actStateNo => #StationInfo.StateNo,
                               info_actStateDescription => #StationInfo.StateDescription,
                               info_errorCode => #StationInfo.ErrorCode,
                               info_warningCode => #StationInfo.WarningCode);
   END_IF;
END_REGION

